KUKA KRL program: MyProgram_242().src

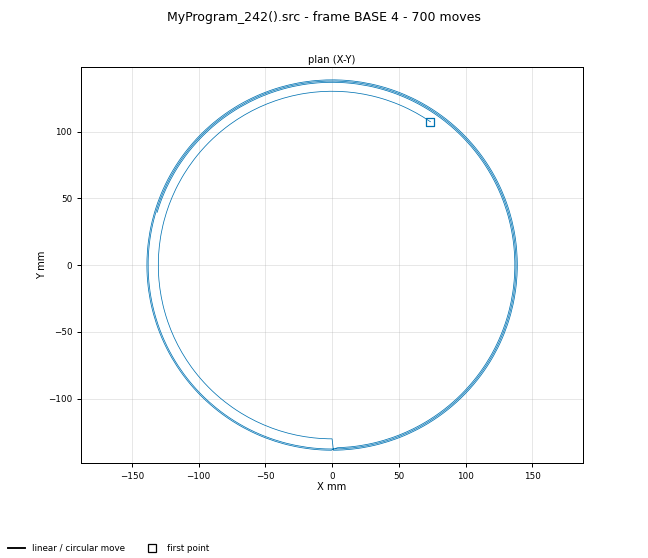
[picture p0: tool path of MyProgram_242().src in frame BASE 4, 700 of 700 moves have a stored position in this frame; points joined in program order, loops and branches not executed]
&ACCESS RVP
&REL 1
&PARAM TEMPLATE = C:\KRC\Roboter\Template\vorgabe
&PARAM EDITMASK = *
DEF MyProgram_242()
; ---- Setting reference (Base) ----
$BASE = BASE_DATA[4]

; --------------------------
; ---- Setting tool (TCP) ----
$TOOL = TOOL_DATA[3]
; --------------------------

$VEL.CP = VEL_APROX_PRINT
Startdeposition()
$VEL.CP = VEL_PRINT
LIN {X 73.6259,Y 107.3159,Z 161,A 55.1179,B 14.0852,C -0.2043,E1 14.1765,E2 754.5488} C_DIS
LIN {X 70.9847,Y 109.081,Z 161,A 56.5627,B 14.0851,C -0.2078,E1 14.1731,E2 753.0982} C_DIS
LIN {X 68.1836,Y 110.8535,Z 161,A 57.9076,B 14.0851,C -0.2066,E1 14.17,E2 751.7664} C_DIS
LIN {X 65.4361,Y 112.4974,Z 161,A 59.3048,B 14.0851,C -0.2083,E1 14.1666,E2 750.3704} C_DIS
LIN {X 62.7519,Y 114.0166,Z 161,A 60.6768,B 14.0851,C -0.2106,E1 14.1633,E2 748.9965} C_DIS
LIN {X 59.8481,Y 115.5669,Z 161,A 62.1112,B 14.0851,C -0.212,E1 14.1597,E2 747.5636} C_DIS
LIN {X 56.9987,Y 116.9979,Z 161,A 63.5064,B 14.085,C -0.2135,E1 14.1562,E2 746.1693} C_DIS
LIN {X 53.5847,Y 118.5997,Z 161,A 65.2897,B 14.085,C -0.2191,E1 14.1517,E2 744.3715} C_DIS
LIN {X 50.1104,Y 120.1079,Z 161,A 66.8675,B 14.085,C -0.2183,E1 14.1476,E2 742.804} C_DIS
LIN {X 46.7383,Y 121.4607,Z 161,A 68.4744,B 14.0849,C -0.2201,E1 14.1434,E2 741.1964} C_DIS
LIN {X 43.7469,Y 122.5698,Z 161,A 69.8364,B 14.0849,C -0.2202,E1 14.1399,E2 739.8394} C_DIS
LIN {X 40.8271,Y 123.5728,Z 161,A 71.1622,B 14.0849,C -0.2204,E1 14.1364,E2 738.5175} C_DIS
LIN {X 37.7836,Y 124.5371,Z 161,A 72.5623,B 14.0849,C -0.2214,E1 14.1327,E2 737.1182} C_DIS
LIN {X 33.9943,Y 125.625,Z 161,A 74.4676,B 14.0848,C -0.2276,E1 14.1275,E2 735.1934} C_DIS
LIN {X 30.0784,Y 126.6195,Z 161,A 76.0649,B 14.0848,C -0.2234,E1 14.1232,E2 733.6176} C_DIS
LIN {X 26.8751,Y 127.3386,Z 161,A 77.4994,B 14.0848,C -0.2239,E1 14.1193,E2 732.1847} C_DIS
LIN {X 23.8559,Y 127.9386,Z 161,A 78.9842,B 14.0848,C -0.2283,E1 14.1152,E2 730.6852} C_DIS
LIN {X 19.9821,Y 128.5993,Z 161,A 80.3539,B 14.0849,C -0.2187,E1 14.1115,E2 729.3576} C_DIS
LIN {X 17.4097,Y 128.9737,Z 161,A 81.7136,B 14.0849,C -0.2252,E1 14.1077,E2 727.9733} C_DIS
LIN {X 14.242,Y 129.3613,Z 161,A 83.119,B 14.0849,C -0.2256,E1 14.1038,E2 726.5684} C_DIS
LIN {X 11.1666,Y 129.6628,Z 161,A 84.5021,B 14.0848,C -0.2265,E1 14.0999,E2 725.1832} C_DIS
LIN {X 7.9833,Y 129.8975,Z 161,A 85.9176,B 14.0848,C -0.2269,E1 14.096,E2 723.767} C_DIS
LIN {X 4.786,Y 130.0549,Z 161,A 87.3094,B 14.0848,C -0.2265,E1 14.0921,E2 722.3779} C_DIS
LIN {X 1.4943,Y 130.1358,Z 161,A 88.733,B 14.0848,C -0.2257,E1 14.0882,E2 720.9579} C_DIS
LIN {X -1.5932,Y 130.1342,Z 161,A 90.1699,B 14.0848,C -0.2278,E1 14.0841,E2 719.5127} C_DIS
LIN {X -5.1925,Y 130.039,Z 161,A 91.6534,B 14.0848,C -0.2246,E1 14.08,E2 718.0418} C_DIS
LIN {X -8.0856,Y 129.8912,Z 161,A 92.9819,B 14.0848,C -0.2258,E1 14.0763,E2 716.7078} C_DIS
LIN {X -11.2683,Y 129.6542,Z 161,A 94.372,B 14.0848,C -0.2249,E1 14.0724,E2 715.3202} C_DIS
LIN {X -14.4438,Y 129.3396,Z 161,A 95.7808,B 14.0848,C -0.2245,E1 14.0685,E2 713.9118} C_DIS
LIN {X -17.6126,Y 128.9471,Z 161,A 97.3138,B 14.0848,C -0.2273,E1 14.0642,E2 712.365} C_DIS
LIN {X -20.6298,Y 128.499,Z 161,A 98.5394,B 14.0848,C -0.2233,E1 14.0609,E2 711.1539} C_DIS
LIN {X -23.9131,Y 127.9277,Z 161,A 100.0038,B 14.0848,C -0.2224,E1 14.0569,E2 709.6908} C_DIS
LIN {X -27.4493,Y 127.2146,Z 161,A 101.5101,B 14.0849,C -0.219,E1 14.0528,E2 708.1949} C_DIS
LIN {X -30.151,Y 126.602,Z 161,A 102.8492,B 14.0849,C -0.2214,E1 14.0491,E2 706.843} C_DIS
LIN {X -33.2702,Y 125.818,Z 161,A 104.3001,B 14.0849,C -0.2212,E1 14.0452,E2 705.3891} C_DIS
LIN {X -36.3399,Y 124.9659,Z 161,A 105.6665,B 14.0849,C -0.2189,E1 14.0415,E2 704.0279} C_DIS
LIN {X -39.3872,Y 124.0391,Z 161,A 107.073,B 14.0849,C -0.2177,E1 14.0378,E2 702.622} C_DIS
LIN {X -42.3168,Y 123.0707,Z 161,A 108.4441,B 14.0849,C -0.2166,E1 14.0341,E2 701.2507} C_DIS
LIN {X -45.3437,Y 121.9879,Z 161,A 109.885,B 14.0849,C -0.2157,E1 14.0304,E2 699.8079} C_DIS
LIN {X -48.4193,Y 120.7999,Z 161,A 111.3149,B 14.0849,C -0.2134,E1 14.0267,E2 698.3819} C_DIS
LIN {X -51.3848,Y 119.5686,Z 161,A 112.7332,B 14.085,C -0.2118,E1 14.023,E2 696.9643} C_DIS
LIN {X -54.2001,Y 118.3196,Z 161,A 114.1986,B 14.085,C -0.213,E1 14.0193,E2 695.4875} C_DIS
LIN {X -57.0785,Y 116.9586,Z 161,A 115.5012,B 14.085,C -0.2084,E1 14.016,E2 694.1977} C_DIS
LIN {X -59.9209,Y 115.5287,Z 161,A 116.919,B 14.085,C -0.2068,E1 14.0125,E2 692.7793} C_DIS
LIN {X -62.7222,Y 114.0331,Z 161,A 118.3262,B 14.0851,C -0.2049,E1 14.009,E2 691.3724} C_DIS
LIN {X -65.5265,Y 112.4451,Z 161,A 119.7877,B 14.0851,C -0.2038,E1 14.0055,E2 689.9074} C_DIS
LIN {X -68.3598,Y 110.7454,Z 161,A 121.3351,B 14.0851,C -0.2039,E1 14.0018,E2 688.3507} C_DIS
LIN {X -71.0666,Y 109.0278,Z 161,A 122.6353,B 14.0852,C -0.1986,E1 13.9988,E2 687.0649} C_DIS
LIN {X -74.0034,Y 107.0567,Z 161,A 124.1527,B 14.0852,C -0.1948,E1 13.9953,E2 685.5537} C_DIS
LIN {X -76.3034,Y 105.4289,Z 161,A 125.5318,B 14.0852,C -0.1962,E1 13.9921,E2 684.1599} C_DIS
LIN {X -79.477,Y 103.0581,Z 161,A 127.3516,B 14.0852,C -0.1949,E1 13.988,E2 682.3333} C_DIS
LIN {X -83.0592,Y 100.193,Z 161,A 129.2786,B 14.0853,C -0.1885,E1 13.9839,E2 680.4192} C_DIS
LIN {X -86.2133,Y 97.4923,Z 161,A 131.2268,B 14.0853,C -0.188,E1 13.9798,E2 678.4592} C_DIS
LIN {X -89.1958,Y 94.7713,Z 161,A 132.9988,B 14.0853,C -0.1841,E1 13.9761,E2 676.6899} C_DIS
LIN {X -92.2874,Y 91.7633,Z 161,A 134.8732,B 14.0855,C -0.1793,E1 13.9724,E2 674.8205} C_DIS
LIN {X -95.3546,Y 88.5719,Z 161,A 136.7631,B 14.0855,C -0.1734,E1 13.9688,E2 672.9397} C_DIS
LIN {X -98.0222,Y 85.6103,Z 161,A 138.665,B 14.0855,C -0.1732,E1 13.9653,E2 671.0229} C_DIS
LIN {X -101.0689,Y 81.9919,Z 161,A 140.6548,B 14.0856,C -0.1659,E1 13.9618,E2 669.0464} C_DIS
LIN {X -103.5133,Y 78.883,Z 161,A 142.367,B 14.0856,C -0.1609,E1 13.9588,E2 667.3397} C_DIS
LIN {X -105.4767,Y 76.2375,Z 161,A 143.8459,B 14.0857,C -0.158,E1 13.9564,E2 665.8592} C_DIS
LIN {X -107.3136,Y 73.6292,Z 161,A 145.2685,B 14.0857,C -0.155,E1 13.9541,E2 664.4363} C_DIS
LIN {X -109.0913,Y 70.9688,Z 161,A 146.6792,B 14.0857,C -0.1514,E1 13.952,E2 663.0271} C_DIS
LIN {X -110.8493,Y 68.1904,Z 161,A 148.1401,B 14.0858,C -0.148,E1 13.9498,E2 661.5664} C_DIS
LIN {X -112.4949,Y 65.4403,Z 161,A 149.6242,B 14.0858,C -0.1462,E1 13.9477,E2 660.0757} C_DIS
LIN {X -114.1557,Y 62.4979,Z 161,A 151.0218,B 14.0858,C -0.1399,E1 13.9458,E2 658.6904} C_DIS
LIN {X -115.5768,Y 59.8291,Z 161,A 152.4245,B 14.0859,C -0.1382,E1 13.944,E2 657.2811} C_DIS
LIN {X -117.0061,Y 56.9822,Z 161,A 153.8389,B 14.0859,C -0.1346,E1 13.9422,E2 655.8671} C_DIS
LIN {X -118.489,Y 53.8322,Z 161,A 155.3666,B 14.0859,C -0.1303,E1 13.9404,E2 654.3419} C_DIS
LIN {X -119.6145,Y 51.2786,Z 161,A 156.6245,B 14.086,C -0.1276,E1 13.939,E2 653.0822} C_DIS
LIN {X -120.8349,Y 48.3325,Z 161,A 158.0533,B 14.086,C -0.1243,E1 13.9375,E2 651.6522} C_DIS
LIN {X -122.019,Y 45.2606,Z 161,A 159.5081,B 14.086,C -0.1203,E1 13.9361,E2 650.1987} C_DIS
LIN {X -123.0645,Y 42.3345,Z 161,A 160.8894,B 14.0861,C -0.1167,E1 13.9348,E2 648.8176} C_DIS
LIN {X -124.0689,Y 39.294,Z 161,A 162.312,B 14.0861,C -0.113,E1 13.9336,E2 647.3953} C_DIS
LIN {X -124.9947,Y 36.2415,Z 161,A 163.8195,B 14.0861,C -0.1115,E1 13.9324,E2 645.8775} C_DIS
LIN {X -125.8456,Y 33.1671,Z 161,A 165.1509,B 14.0861,C -0.1056,E1 13.9315,E2 644.5565} C_DIS
LIN {X -126.6208,Y 30.0728,Z 161,A 166.5675,B 14.0862,C -0.1018,E1 13.9305,E2 643.1402} C_DIS
LIN {X -127.3728,Y 26.717,Z 161,A 168.0921,B 14.0862,C -0.0976,E1 13.9296,E2 641.6164} C_DIS
LIN {X -127.9447,Y 23.8242,Z 161,A 169.4945,B 14.0862,C -0.0964,E1 13.9289,E2 640.2034} C_DIS
LIN {X -128.493,Y 20.668,Z 161,A 170.8524,B 14.0862,C -0.0908,E1 13.9283,E2 638.8534} C_DIS
LIN {X -128.973,Y 17.4148,Z 161,A 172.2813,B 14.0863,C -0.0861,E1 13.9277,E2 637.4285} C_DIS
LIN {X -129.3602,Y 14.2523,Z 161,A 173.7018,B 14.0863,C -0.0823,E1 13.9272,E2 636.0076} C_DIS
LIN {X -129.6614,Y 11.1832,Z 161,A 175.1006,B 14.0863,C -0.0793,E1 13.9269,E2 634.6056} C_DIS
LIN {X -129.8984,Y 7.9682,Z 161,A 176.6346,B 14.0863,C -0.078,E1 13.9266,E2 633.0601} C_DIS
LIN {X -130.1053,Y 3.1501,Z 161,A 178.8132,B 14.0863,C -0.073,E1 13.9264,E2 630.8775} C_DIS
LIN {X -130.1443,Y -0.1417,Z 161,A -179.8418,B 14.0864,C -0.066,E1 13.9264,E2 629.5464} C_DIS
LIN {X -130.0999,Y -3.3439,Z 161,A -178.4539,B 14.0864,C -0.0612,E1 13.9264,E2 628.1627} C_DIS
LIN {X -129.9457,Y -7.1863,Z 161,A -176.5128,B 14.0864,C -0.0625,E1 13.9267,E2 626.1947} C_DIS
LIN {X -129.6591,Y -11.2103,Z 161,A -174.791,B 14.0864,C -0.0558,E1 13.9271,E2 624.4813} C_DIS
LIN {X -129.3395,Y -14.444,Z 161,A -173.4951,B 14.0864,C -0.0481,E1 13.9275,E2 623.2028} C_DIS
LIN {X -128.9453,Y -17.6265,Z 161,A -172.0481,B 14.0865,C -0.0448,E1 13.928,E2 621.7532} C_DIS
LIN {X -128.4921,Y -20.6737,Z 161,A -170.6312,B 14.0865,C -0.0424,E1 13.9286,E2 620.3307} C_DIS
LIN {X -127.9276,Y -23.9136,Z 161,A -169.2425,B 14.0865,C -0.0367,E1 13.9293,E2 618.9505} C_DIS
LIN {X -127.3036,Y -27.0372,Z 161,A -167.7841,B 14.0865,C -0.034,E1 13.9301,E2 617.487} C_DIS
LIN {X -126.5963,Y -30.1746,Z 161,A -166.3629,B 14.0865,C -0.0301,E1 13.931,E2 616.0666} C_DIS
LIN {X -125.8186,Y -33.2682,Z 161,A -164.8112,B 14.0865,C -0.0298,E1 13.9321,E2 614.4991} C_DIS
LIN {X -124.5105,Y -37.8707,Z 161,A -162.6746,B 14.0865,C -0.0246,E1 13.9338,E2 612.3611} C_DIS
LIN {X -123.0627,Y -42.3397,Z 161,A -160.5991,B 14.0865,C -0.019,E1 13.9356,E2 610.2868} C_DIS
LIN {X -121.9873,Y -45.3452,Z 161,A -159.2767,B 14.0865,C -0.013,E1 13.9369,E2 608.9755} C_DIS
LIN {X -120.796,Y -48.4289,Z 161,A -157.8194,B 14.0865,C -0.009,E1 13.9384,E2 607.5193} C_DIS
LIN {X -119.4274,Y -51.7114,Z 161,A -156.3496,B 14.0865,C -0.0023,E1 13.94,E2 606.0621} C_DIS
LIN {X -118.3288,Y -54.1803,Z 161,A -155.0611,B 14.0865,C -0.0017,E1 13.9415,E2 604.7631} C_DIS
LIN {X -116.9719,Y -57.0514,Z 161,A -153.6354,B 14.0865,C 0.0013,E1 13.9432,E2 603.3354} C_DIS
LIN {X -115.5201,Y -59.9372,Z 161,A -152.2025,B 14.0865,C 0.0047,E1 13.945,E2 601.9025} C_DIS
LIN {X -114.0169,Y -62.7514,Z 161,A -150.793,B 14.0865,C 0.0082,E1 13.9469,E2 600.4936} C_DIS
LIN {X -112.4447,Y -65.5272,Z 161,A -149.2073,B 14.0865,C 0.0071,E1 13.9492,E2 598.8876} C_DIS
LIN {X -110.6283,Y -68.5486,Z 161,A -147.8508,B 14.0865,C 0.016,E1 13.9511,E2 597.5554} C_DIS
LIN {X -109.0315,Y -71.0609,Z 161,A -146.4787,B 14.0865,C 0.0176,E1 13.9532,E2 596.1769} C_DIS
LIN {X -107.2589,Y -73.709,Z 161,A -145.0641,B 14.0865,C 0.0207,E1 13.9554,E2 594.762} C_DIS
LIN {X -105.4136,Y -76.3247,Z 161,A -143.6468,B 14.0865,C 0.0238,E1 13.9577,E2 593.3447} C_DIS
LIN {X -103.0905,Y -79.4352,Z 161,A -141.7683,B 14.0865,C 0.0233,E1 13.9609,E2 591.4474} C_DIS
LIN {X -100.5997,Y -82.5666,Z 161,A -140.0952,B 14.0865,C 0.0296,E1 13.9638,E2 589.7859} C_DIS
LIN {X -97.9974,Y -85.6387,Z 161,A -138.3713,B 14.0865,C 0.0347,E1 13.9669,E2 588.0687} C_DIS
LIN {X -95.8775,Y -88.0056,Z 161,A -136.798,B 14.0865,C 0.0331,E1 13.9699,E2 586.4756} C_DIS
LIN {X -92.6228,Y -91.4257,Z 161,A -134.8322,B 14.0865,C 0.0404,E1 13.9737,E2 584.5242} C_DIS
LIN {X -89.7209,Y -94.2747,Z 161,A -132.8894,B 14.0865,C 0.0398,E1 13.9777,E2 582.5643} C_DIS
LIN {X -86.8005,Y -96.9698,Z 161,A -131.2805,B 14.0865,C 0.047,E1 13.981,E2 580.9727} C_DIS
LIN {X -83.8113,Y -99.5649,Z 161,A -129.3858,B 14.0865,C 0.0461,E1 13.985,E2 579.0608} C_DIS
LIN {X -80.1295,Y -102.5517,Z 161,A -127.4162,B 14.0865,C 0.0529,E1 13.9893,E2 577.1058} C_DIS
LIN {X -77.5216,Y -104.5367,Z 161,A -125.9765,B 14.0865,C 0.0554,E1 13.9925,E2 575.667} C_DIS
LIN {X -74.9412,Y -106.4016,Z 161,A -124.5698,B 14.0865,C 0.0576,E1 13.9957,E2 574.2602} C_DIS
LIN {X -71.6886,Y -108.6197,Z 161,A -122.6855,B 14.0865,C 0.0562,E1 14.0001,E2 572.3583} C_DIS
LIN {X -68.1778,Y -110.8571,Z 161,A -120.9872,B 14.0865,C 0.0625,E1 14.0041,E2 570.6765} C_DIS
LIN {X -65.4414,Y -112.4943,Z 161,A -119.5778,B 14.0865,C 0.0643,E1 14.0075,E2 569.2667} C_DIS
LIN {X -62.7563,Y -114.0142,Z 161,A -118.1916,B 14.0865,C 0.0654,E1 14.0109,E2 567.8774} C_DIS
LIN {X -59.8522,Y -115.5647,Z 161,A -116.7433,B 14.0865,C 0.0672,E1 14.0144,E2 566.4294} C_DIS
LIN {X -57.0023,Y -116.9962,Z 161,A -115.3347,B 14.0865,C 0.0688,E1 14.018,E2 565.0203} C_DIS
LIN {X -53.636,Y -118.5767,Z 161,A -113.7967,B 14.0864,C 0.0734,E1 14.0218,E2 563.4942} C_DIS
LIN {X -51.2692,Y -119.6186,Z 161,A -112.5522,B 14.0864,C 0.0716,E1 14.0251,E2 562.2372} C_DIS
LIN {X -47.7588,Y -121.064,Z 161,A -110.9356,B 14.0864,C 0.0748,E1 14.0292,E2 560.6271} C_DIS
LIN {X -44.8477,Y -122.173,Z 161,A -109.519,B 14.0864,C 0.0748,E1 14.0329,E2 559.2051} C_DIS
LIN {X -42.3399,Y -123.0627,Z 161,A -108.3263,B 14.0864,C 0.0752,E1 14.0361,E2 558.0097} C_DIS
LIN {X -39.3122,Y -124.063,Z 161,A -106.9169,B 14.0864,C 0.0762,E1 14.0398,E2 556.5995} C_DIS
LIN {X -36.2456,Y -124.9935,Z 161,A -105.4997,B 14.0864,C 0.077,E1 14.0436,E2 555.1814} C_DIS
LIN {X -33.1768,Y -125.843,Z 161,A -104.1015,B 14.0864,C 0.078,E1 14.0474,E2 553.7834} C_DIS
LIN {X -30.0897,Y -126.6168,Z 161,A -102.6988,B 14.0864,C 0.0787,E1 14.0512,E2 552.3803} C_DIS
LIN {X -26.8938,Y -127.3346,Z 161,A -101.262,B 14.0864,C 0.0796,E1 14.0551,E2 550.9438} C_DIS
LIN {X -23.2646,Y -128.0466,Z 161,A -99.7802,B 14.0864,C 0.0844,E1 14.0592,E2 549.4791} C_DIS
LIN {X -20.6714,Y -128.4925,Z 161,A -98.4478,B 14.0864,C 0.0799,E1 14.0629,E2 548.1257} C_DIS
LIN {X -17.411,Y -128.9735,Z 161,A -97.0294,B 14.0864,C 0.0812,E1 14.0668,E2 546.7106} C_DIS
LIN {X -14.2422,Y -129.3612,Z 161,A -95.4636,B 14.0864,C 0.0769,E1 14.0712,E2 545.1252} C_DIS
LIN {X -9.5785,Y -129.7896,Z 161,A -93.5043,B 14.0864,C 0.08,E1 14.0766,E2 543.1773} C_DIS
LIN {X -6.2811,Y -129.9912,Z 161,A -92.1053,B 14.0864,C 0.0817,E1 14.0805,E2 541.7844} C_DIS
LIN {X -3.0902,Y -130.107,Z 161,A -90.699,B 14.0864,C 0.0816,E1 14.0844,E2 540.3774} C_DIS
LIN {X -0.0064,Y -130.1446,Z 161,A -89.2963,B 14.0864,C 0.0801,E1 14.0884,E2 538.9687} C_DIS
LIN {X -0.0064,Y -130.1446,Z 161,A -89.2963,B 14.0864,C 0.0801,E1 14.0884,E2 538.9687} C_DIS
Enddeposition()
LIN {X 0.9753,Y -138.6804,Z 162,A -92.6437,B 24.9722,C -1.2174,E1 25.001,E2 539.3993} C_DIS
Startdeposition()
$VEL.CP = VEL_PRINT
LIN {X 3.7085,Y -138.6375,Z 162,A -90.9723,B 24.9708,C -1.2478,E1 25.0059,E2 537.6562} C_DIS
LIN {X 8.2859,Y -138.4394,Z 162,A -88.9916,B 24.9706,C -1.2535,E1 25.0114,E2 535.6628} C_DIS
LIN {X 14.8199,Y -137.8928,Z 162,A -86.3827,B 24.9708,C -1.2494,E1 25.0186,E2 533.0653} C_DIS
LIN {X 19.2083,Y -137.3508,Z 162,A -84.5954,B 24.9708,C -1.2483,E1 25.0236,E2 531.2819} C_DIS
LIN {X 22.4873,Y -136.852,Z 162,A -83.2381,B 24.9708,C -1.2486,E1 25.0273,E2 529.9251} C_DIS
LIN {X 28.0328,Y -135.8246,Z 162,A -80.8102,B 24.9704,C -1.2562,E1 25.034,E2 527.4823} C_DIS
LIN {X 32.1897,Y -134.8997,Z 162,A -79.1481,B 24.9706,C -1.2524,E1 25.0385,E2 525.8314} C_DIS
LIN {X 35.5715,Y -134.0473,Z 162,A -77.6983,B 24.9706,C -1.2544,E1 25.0424,E2 524.3791} C_DIS
LIN {X 39.11,Y -133.0579,Z 162,A -76.2619,B 24.9706,C -1.2515,E1 25.0463,E2 522.9519} C_DIS
LIN {X 42.0399,Y -132.1614,Z 162,A -75.0069,B 24.9706,C -1.2525,E1 25.0496,E2 521.697} C_DIS
LIN {X 45.6855,Y -130.9461,Z 162,A -73.6635,B 24.9712,C -1.2407,E1 25.0531,E2 520.3841} C_DIS
LIN {X 48.0279,Y -130.1065,Z 162,A -72.2874,B 24.9702,C -1.2618,E1 25.0568,E2 518.9609} C_DIS
LIN {X 51.3498,Y -128.831,Z 162,A -70.9235,B 24.9704,C -1.2579,E1 25.0603,E2 517.6094} C_DIS
LIN {X 54.6499,Y -127.4657,Z 162,A -69.429,B 24.9702,C -1.2612,E1 25.0642,E2 516.1105} C_DIS
LIN {X 57.9984,Y -125.9769,Z 162,A -67.9996,B 24.9703,C -1.2587,E1 25.0678,E2 514.6904} C_DIS
LIN {X 61.0435,Y -124.53,Z 162,A -66.5311,B 24.97,C -1.2654,E1 25.0715,E2 513.2101} C_DIS
LIN {X 63.9672,Y -123.0547,Z 162,A -65.1072,B 24.9697,C -1.2718,E1 25.0751,E2 511.775} C_DIS
LIN {X 67.9591,Y -120.8968,Z 162,A -63.229,B 24.9695,C -1.2754,E1 25.0797,E2 509.8938} C_DIS
LIN {X 71.8296,Y -118.6381,Z 162,A -61.3598,B 24.9693,C -1.2799,E1 25.0842,E2 508.0197} C_DIS
LIN {X 75.7781,Y -116.1561,Z 162,A -59.4156,B 24.9691,C -1.2847,E1 25.0888,E2 506.0703} C_DIS
LIN {X 79.6326,Y -113.5485,Z 162,A -57.504,B 24.9689,C -1.2881,E1 25.0932,E2 504.1573} C_DIS
LIN {X 83.0656,Y -111.0616,Z 162,A -55.7626,B 24.9688,C -1.2913,E1 25.0971,E2 502.4146} C_DIS
LIN {X 86.6721,Y -108.2708,Z 162,A -53.9067,B 24.9686,C -1.2939,E1 25.1011,E2 500.5595} C_DIS
LIN {X 90.2073,Y -105.3436,Z 162,A -52.1152,B 24.9687,C -1.2922,E1 25.105,E2 498.7788} C_DIS
LIN {X 93.3673,Y -102.5528,Z 162,A -50.2808,B 24.9683,C -1.3018,E1 25.1088,E2 496.9292} C_DIS
LIN {X 96.8454,Y -99.2752,Z 162,A -48.3436,B 24.9681,C -1.3045,E1 25.1127,E2 494.9937} C_DIS
LIN {X 99.9045,Y -96.1962,Z 162,A -46.6208,B 24.9681,C -1.305,E1 25.1161,E2 493.2772} C_DIS
LIN {X 102.8585,Y -93.0304,Z 162,A -44.7439,B 24.9676,C -1.3148,E1 25.1196,E2 491.3854} C_DIS
LIN {X 105.9921,Y -89.4444,Z 162,A -42.8137,B 24.9675,C -1.3178,E1 25.1231,E2 489.4567} C_DIS
LIN {X 108.8664,Y -85.9226,Z 162,A -40.9278,B 24.9672,C -1.3235,E1 25.1264,E2 487.5664} C_DIS
LIN {X 111.3769,Y -82.6421,Z 162,A -39.2245,B 24.967,C -1.328,E1 25.1293,E2 485.8604} C_DIS
LIN {X 113.7244,Y -79.3806,Z 162,A -37.6296,B 24.967,C -1.329,E1 25.1319,E2 484.2711} C_DIS
LIN {X 116.1586,Y -75.7744,Z 162,A -35.8119,B 24.9666,C -1.3353,E1 25.1347,E2 482.4473} C_DIS
LIN {X 118.5147,Y -72.0336,Z 162,A -34.0007,B 24.9664,C -1.3398,E1 25.1373,E2 480.6348} C_DIS
LIN {X 120.7254,Y -68.2641,Z 162,A -32.2065,B 24.9661,C -1.3446,E1 25.1398,E2 478.8387} C_DIS
LIN {X 122.8089,Y -64.4352,Z 162,A -30.5511,B 24.9663,C -1.3416,E1 25.142,E2 477.199} C_DIS
LIN {X 124.191,Y -61.7308,Z 162,A -29.3366,B 24.9663,C -1.3431,E1 25.1435,E2 475.9875} C_DIS
LIN {X 125.746,Y -58.4976,Z 162,A -27.988,B 24.9663,C -1.3399,E1 25.1451,E2 474.6537} C_DIS
LIN {X 127.389,Y -54.8273,Z 162,A -26.1614,B 24.9656,C -1.3547,E1 25.1472,E2 472.802} C_DIS
LIN {X 128.7705,Y -51.5,Z 162,A -24.6262,B 24.9652,C -1.3622,E1 25.1488,E2 471.2577} C_DIS
LIN {X 130.3355,Y -47.4,Z 162,A -22.8953,B 24.9652,C -1.3632,E1 25.1505,E2 469.5342} C_DIS
LIN {X 131.3138,Y -44.6245,Z 162,A -21.5185,B 24.9645,C -1.3765,E1 25.1518,E2 468.1337} C_DIS
LIN {X 132.6699,Y -40.4067,Z 162,A -19.8106,B 24.9645,C -1.3753,E1 25.1532,E2 466.4384} C_DIS
LIN {X 133.7855,Y -36.5526,Z 162,A -18.0491,B 24.964,C -1.3868,E1 25.1545,E2 464.66} C_DIS
LIN {X 135.5398,Y -29.3766,Z 162,A -15.2875,B 24.9643,C -1.3797,E1 25.1563,E2 461.931} C_DIS
LIN {X 136.5038,Y -24.5099,Z 162,A -13.0623,B 24.9635,C -1.3968,E1 25.1575,E2 459.6785} C_DIS
LIN {X 137.461,Y -18.4024,Z 162,A -10.5107,B 24.963,C -1.4051,E1 25.1586,E2 457.1223} C_DIS
LIN {X 137.9164,Y -14.6005,Z 162,A -9.0149,B 24.963,C -1.4053,E1 25.159,E2 455.6348} C_DIS
LIN {X 138.2749,Y -10.6987,Z 162,A -7.3449,B 24.9626,C -1.4137,E1 25.1594,E2 453.9549} C_DIS
LIN {X 138.4663,Y -7.8494,Z 162,A -6.0652,B 24.962,C -1.4235,E1 25.1596,E2 452.6597} C_DIS
LIN {X 138.6555,Y -3.0458,Z 162,A -4.1721,B 24.962,C -1.4247,E1 25.1598,E2 450.7752} C_DIS
LIN {X 138.6846,Y 0.9336,Z 162,A -2.5259,B 24.9617,C -1.4303,E1 25.1598,E2 449.1256} C_DIS
LIN {X 138.5957,Y 5.0433,Z 162,A -0.7011,B 24.961,C -1.4434,E1 25.1596,E2 447.2808} C_DIS
LIN {X 138.1484,Y 12.2225,Z 162,A 2.1078,B 24.961,C -1.4436,E1 25.159,E2 444.4881} C_DIS
LIN {X 137.7591,Y 16.0201,Z 162,A 3.6244,B 24.9609,C -1.4452,E1 25.1586,E2 442.9766} C_DIS
LIN {X 137.2957,Y 19.5936,Z 162,A 5.4378,B 24.9596,C -1.4692,E1 25.1579,E2 441.1174} C_DIS
LIN {X 136.6815,Y 23.5089,Z 162,A 6.7441,B 24.9603,C -1.455,E1 25.1573,E2 439.8522} C_DIS
LIN {X 136.0133,Y 27.1056,Z 162,A 8.2737,B 24.96,C -1.461,E1 25.1565,E2 438.3175} C_DIS
LIN {X 135.2956,Y 30.4839,Z 162,A 9.586,B 24.9601,C -1.4588,E1 25.1557,E2 437.0179} C_DIS
LIN {X 134.5402,Y 33.6623,Z 162,A 10.9233,B 24.9599,C -1.4624,E1 25.1548,E2 435.6799} C_DIS
LIN {X 133.7126,Y 36.8137,Z 162,A 12.2469,B 24.9598,C -1.4654,E1 25.1538,E2 434.3569} C_DIS
LIN {X 132.8113,Y 39.9448,Z 162,A 13.6471,B 24.9594,C -1.4727,E1 25.1527,E2 432.9474} C_DIS
LIN {X 131.8109,Y 43.1321,Z 162,A 14.9339,B 24.9594,C -1.4716,E1 25.1516,E2 431.6707} C_DIS
LIN {X 130.6246,Y 46.598,Z 162,A 16.4084,B 24.9594,C -1.474,E1 25.1503,E2 430.1988} C_DIS
LIN {X 129.3548,Y 50.0134,Z 162,A 18.0698,B 24.9585,C -1.4876,E1 25.1486,E2 428.5144} C_DIS
LIN {X 127.9962,Y 53.3939,Z 162,A 19.4247,B 24.9588,C -1.4834,E1 25.1472,E2 427.177} C_DIS
LIN {X 126.8443,Y 56.0786,Z 162,A 20.6478,B 24.9585,C -1.4879,E1 25.1458,E2 425.9499} C_DIS
LIN {X 125.4423,Y 59.1495,Z 162,A 22.1319,B 24.958,C -1.4972,E1 25.1441,E2 424.452} C_DIS
LIN {X 123.9038,Y 62.3077,Z 162,A 23.4532,B 24.9582,C -1.4938,E1 25.1424,E2 423.1457} C_DIS
LIN {X 122.0968,Y 65.779,Z 162,A 25.225,B 24.9574,C -1.5074,E1 25.1401,E2 421.3512} C_DIS
LIN {X 119.8214,Y 69.8389,Z 162,A 27.1533,B 24.9571,C -1.5131,E1 25.1374,E2 419.4195} C_DIS
LIN {X 117.384,Y 73.8614,Z 162,A 28.9985,B 24.9571,C -1.5127,E1 25.1347,E2 417.5846} C_DIS
LIN {X 115.1906,Y 77.2377,Z 162,A 30.6508,B 24.9569,C -1.5165,E1 25.1322,E2 415.9316} C_DIS
LIN {X 112.8106,Y 80.6736,Z 162,A 32.3991,B 24.9566,C -1.5222,E1 25.1294,E2 414.1783} C_DIS
LIN {X 110.2402,Y 84.1521,Z 162,A 34.1841,B 24.9563,C -1.5266,E1 25.1264,E2 412.3914} C_DIS
LIN {X 107.5398,Y 87.5769,Z 162,A 35.9758,B 24.9561,C -1.5305,E1 25.1232,E2 410.5989} C_DIS
LIN {X 104.687,Y 90.968,Z 162,A 37.8485,B 24.9557,C -1.5373,E1 25.1198,E2 408.7186} C_DIS
LIN {X 101.5212,Y 94.4877,Z 162,A 39.7526,B 24.9557,C -1.5389,E1 25.1162,E2 406.8193} C_DIS
LIN {X 98.4714,Y 97.662,Z 162,A 41.5766,B 24.9554,C -1.5432,E1 25.1127,E2 404.9928} C_DIS
LIN {X 95.1807,Y 100.8717,Z 162,A 43.4532,B 24.9552,C -1.546,E1 25.1089,E2 403.1173} C_DIS
LIN {X 91.9435,Y 103.831,Z 162,A 45.1593,B 24.9553,C -1.5438,E1 25.1054,E2 401.4234} C_DIS
LIN {X 88.9102,Y 106.4403,Z 162,A 46.9207,B 24.9548,C -1.5532,E1 25.1016,E2 399.6466} C_DIS
LIN {X 85.4258,Y 109.2566,Z 162,A 48.7513,B 24.9547,C -1.5556,E1 25.0976,E2 397.8172} C_DIS
LIN {X 81.956,Y 111.8826,Z 162,A 50.5337,B 24.9545,C -1.558,E1 25.0936,E2 396.0354} C_DIS
LIN {X 78.3975,Y 114.4042,Z 162,A 52.2951,B 24.9545,C -1.5589,E1 25.0896,E2 394.2781} C_DIS
LIN {X 74.835,Y 116.7656,Z 162,A 54.0846,B 24.9542,C -1.5631,E1 25.0854,E2 392.4844} C_DIS
LIN {X 71.4071,Y 118.8936,Z 162,A 55.799,B 24.9539,C -1.5684,E1 25.0813,E2 390.763} C_DIS
LIN {X 67.3342,Y 121.2461,Z 162,A 57.7096,B 24.9539,C -1.5694,E1 25.0766,E2 388.8556} C_DIS
LIN {X 63.1987,Y 123.4502,Z 162,A 59.5084,B 24.9541,C -1.5644,E1 25.0722,E2 387.0738} C_DIS
LIN {X 60.1258,Y 124.9758,Z 162,A 61.0447,B 24.9536,C -1.5728,E1 25.0683,E2 385.5215} C_DIS
LIN {X 54.0838,Y 127.7081,Z 162,A 63.7749,B 24.9535,C -1.5755,E1 25.0614,E2 382.7917} C_DIS
LIN {X 50.8184,Y 129.0419,Z 162,A 65.0541,B 24.954,C -1.5671,E1 25.0581,E2 381.5354} C_DIS
LIN {X 47.3828,Y 130.3417,Z 162,A 66.5859,B 24.9539,C -1.5694,E1 25.0541,E2 380.0014} C_DIS
LIN {X 44.0908,Y 131.4916,Z 162,A 68.0823,B 24.9536,C -1.5737,E1 25.0501,E2 378.4976} C_DIS
LIN {X 40.3711,Y 132.6808,Z 162,A 69.7223,B 24.9534,C -1.5765,E1 25.0457,E2 376.8539} C_DIS
LIN {X 36.2698,Y 133.8611,Z 162,A 71.4565,B 24.9534,C -1.5761,E1 25.0411,E2 375.1235} C_DIS
LIN {X 33.1096,Y 134.6779,Z 162,A 72.7978,B 24.9534,C -1.5766,E1 25.0375,E2 373.7832} C_DIS
LIN {X 29.5481,Y 135.5027,Z 162,A 74.3494,B 24.9532,C -1.5797,E1 25.0332,E2 372.2263} C_DIS
LIN {X 22.0964,Y 136.9172,Z 162,A 77.6119,B 24.9528,C -1.588,E1 25.0242,E2 368.9478} C_DIS
LIN {X 18.3128,Y 137.4728,Z 162,A 79.0783,B 24.9531,C -1.5822,E1 25.0202,E2 367.4964} C_DIS
LIN {X 15.3307,Y 137.8378,Z 162,A 80.4516,B 24.9527,C -1.5896,E1 25.0163,E2 366.1064} C_DIS
LIN {X 10.2761,Y 138.3058,Z 162,A 82.2843,B 24.9535,C -1.5753,E1 25.0113,E2 364.3087} C_DIS
LIN {X 6.9774,Y 138.5113,Z 162,A 83.8133,B 24.953,C -1.5843,E1 25.007,E2 362.759} C_DIS
LIN {X 1.7495,Y 138.6771,Z 162,A 86.066,B 24.9527,C -1.589,E1 25.0007,E2 360.4956} C_DIS
LIN {X -4.377,Y 138.6189,Z 162,A 88.4104,B 24.9533,C -1.5782,E1 24.9942,E2 358.1767} C_DIS
LIN {X -8.2135,Y 138.4439,Z 162,A 90.073,B 24.9531,C -1.5817,E1 24.9896,E2 356.5051} C_DIS
LIN {X -11.2796,Y 138.228,Z 162,A 91.3447,B 24.9531,C -1.5812,E1 24.986,E2 355.2341} C_DIS
LIN {X -15.2031,Y 137.8515,Z 162,A 92.9131,B 24.9534,C -1.5771,E1 24.9817,E2 353.6745} C_DIS
LIN {X -21.8317,Y 136.9591,Z 162,A 95.8247,B 24.953,C -1.5832,E1 24.9736,E2 350.746} C_DIS
LIN {X -25.8999,Y 136.2469,Z 162,A 97.3948,B 24.9535,C -1.5746,E1 24.9693,E2 349.1949} C_DIS
LIN {X -29.2592,Y 135.5651,Z 162,A 98.7912,B 24.9537,C -1.5723,E1 24.9655,E2 347.8022} C_DIS
LIN {X -32.4537,Y 134.836,Z 162,A 100.1428,B 24.9537,C -1.5709,E1 24.9619,E2 346.4521} C_DIS
LIN {X -35.5954,Y 134.0409,Z 162,A 101.4816,B 24.9538,C -1.5695,E1 24.9582,E2 345.1146} C_DIS
LIN {X -38.5099,Y 133.2336,Z 162,A 102.8193,B 24.9536,C -1.5729,E1 24.9546,E2 343.7668} C_DIS
LIN {X -42.4162,Y 132.0412,Z 162,A 104.4798,B 24.9538,C -1.5694,E1 24.9502,E2 342.1116} C_DIS
LIN {X -46.2608,Y 130.7462,Z 162,A 106.2062,B 24.9538,C -1.57,E1 24.9456,E2 340.3806} C_DIS
LIN {X -52.9314,Y 128.1894,Z 162,A 109.1368,B 24.9541,C -1.5647,E1 24.938,E2 337.4561} C_DIS
LIN {X -55.93,Y 126.9108,Z 162,A 110.4245,B 24.9544,C -1.5596,E1 24.9348,E2 336.1776} C_DIS
LIN {X -59.4666,Y 125.2908,Z 162,A 112.0823,B 24.9544,C -1.5597,E1 24.9306,E2 334.5153} C_DIS
LIN {X -63.2797,Y 123.4089,Z 162,A 114.0981,B 24.9538,C -1.5705,E1 24.9255,E2 332.4684} C_DIS
LIN {X -66.2568,Y 121.8382,Z 162,A 115.2476,B 24.9547,C -1.5553,E1 24.9227,E2 331.3519} C_DIS
LIN {X -69.8279,Y 119.8278,Z 162,A 117.0058,B 24.9547,C -1.5556,E1 24.9184,E2 329.5877} C_DIS
LIN {X -72.8832,Y 117.9945,Z 162,A 118.5463,B 24.9547,C -1.5564,E1 24.9148,E2 328.0405} C_DIS
LIN {X -76.9712,Y 115.3686,Z 162,A 120.5028,B 24.955,C -1.5498,E1 24.9102,E2 326.0934} C_DIS
LIN {X -80.7672,Y 112.7437,Z 162,A 122.4166,B 24.9552,C -1.5462,E1 24.9058,E2 324.1816} C_DIS
LIN {X -84.3925,Y 110.0564,Z 162,A 124.2857,B 24.9554,C -1.5424,E1 24.9017,E2 322.3147} C_DIS
LIN {X -88.0186,Y 107.1788,Z 162,A 126.1283,B 24.9559,C -1.5345,E1 24.8977,E2 320.4841} C_DIS
LIN {X -91.163,Y 104.5169,Z 162,A 127.9255,B 24.9559,C -1.5355,E1 24.8939,E2 318.6775} C_DIS
LIN {X -94.6537,Y 101.3666,Z 162,A 129.8974,B 24.956,C -1.5324,E1 24.8898,E2 316.7049} C_DIS
LIN {X -98.0615,Y 98.0745,Z 162,A 131.8916,B 24.9562,C -1.5295,E1 24.8858,E2 314.7094} C_DIS
LIN {X -101.3864,Y 94.6324,Z 162,A 133.84,B 24.9565,C -1.523,E1 24.8821,E2 312.768} C_DIS
LIN {X -104.514,Y 91.1663,Z 162,A 135.7797,B 24.9568,C -1.5185,E1 24.8785,E2 310.8303} C_DIS
LIN {X -107.4685,Y 87.6642,Z 162,A 137.6801,B 24.9571,C -1.5138,E1 24.8751,E2 308.9323} C_DIS
LIN {X -110.2583,Y 84.1285,Z 162,A 139.526,B 24.9574,C -1.5079,E1 24.872,E2 307.0916} C_DIS
LIN {X -112.8305,Y 80.6459,Z 162,A 141.1723,B 24.9581,C -1.4955,E1 24.8693,E2 305.4667} C_DIS
LIN {X -114.757,Y 77.8802,Z 162,A 143.0753,B 24.9568,C -1.518,E1 24.8662,E2 303.5009} C_DIS
LIN {X -116.9809,Y 74.4987,Z 162,A 144.8244,B 24.9568,C -1.5171,E1 24.8636,E2 301.7449} C_DIS
LIN {X -119.2774,Y 70.7633,Z 162,A 146.1698,B 24.9585,C -1.4876,E1 24.8618,E2 300.4628} C_DIS
LIN {X -121.0636,Y 67.6623,Z 162,A 147.7337,B 24.9585,C -1.4876,E1 24.8596,E2 298.8908} C_DIS
LIN {X -123.1055,Y 63.8703,Z 162,A 149.5097,B 24.9588,C -1.4821,E1 24.8573,E2 297.1186} C_DIS
LIN {X -124.8322,Y 60.4264,Z 162,A 150.9827,B 24.9595,C -1.4711,E1 24.8555,E2 295.6638} C_DIS
LIN {X -126.4561,Y 56.9466,Z 162,A 152.6326,B 24.9595,C -1.4695,E1 24.8536,E2 294.0088} C_DIS
LIN {X -128.0741,Y 53.2074,Z 162,A 155.2849,B 24.957,C -1.5144,E1 24.8506,E2 291.2346} C_DIS
LIN {X -130.5722,Y 46.7435,Z 162,A 157.2578,B 24.9601,C -1.4591,E1 24.8488,E2 289.3824} C_DIS
LIN {X -132.0016,Y 42.5404,Z 162,A 159.0595,B 24.9605,C -1.4515,E1 24.8472,E2 287.5885} C_DIS
LIN {X -133.1463,Y 38.808,Z 162,A 160.6758,B 24.9608,C -1.4465,E1 24.8459,E2 285.9749} C_DIS
LIN {X -134.0231,Y 35.6622,Z 162,A 162.0097,B 24.9611,C -1.4413,E1 24.845,E2 284.6456} C_DIS
LIN {X -134.7841,Y 32.6691,Z 162,A 163.4131,B 24.961,C -1.4436,E1 24.844,E2 283.2284} C_DIS
LIN {X -135.8024,Y 28.1419,Z 162,A 165.2493,B 24.9615,C -1.4332,E1 24.8429,E2 281.4063} C_DIS
LIN {X -136.5108,Y 24.4708,Z 162,A 166.7998,B 24.9618,C -1.4284,E1 24.8421,E2 279.858} C_DIS
LIN {X -137.0751,Y 21.0822,Z 162,A 168.2225,B 24.962,C -1.4239,E1 24.8415,E2 278.4376} C_DIS
LIN {X -137.5325,Y 17.8573,Z 162,A 169.5741,B 24.9622,C -1.4197,E1 24.841,E2 277.0879} C_DIS
LIN {X -137.9119,Y 14.6426,Z 162,A 170.9259,B 24.9624,C -1.416,E1 24.8406,E2 275.7368} C_DIS
LIN {X -138.2715,Y 10.7463,Z 162,A 172.6664,B 24.9624,C -1.417,E1 24.8402,E2 273.9835} C_DIS
LIN {X -138.6134,Y 4.5475,Z 162,A 175.0613,B 24.9633,C -1.3997,E1 24.8399,E2 271.6154} C_DIS
LIN {X -138.6844,Y -0.9781,Z 162,A 177.4806,B 24.9633,C -1.3991,E1 24.8399,E2 269.183} C_DIS
LIN {X -138.6093,Y -4.6957,Z 162,A 178.9811,B 24.9637,C -1.3921,E1 24.8399,E2 267.6899} C_DIS
LIN {X -138.4586,Y -7.9736,Z 162,A -179.6455,B 24.9639,C -1.3886,E1 24.8401,E2 266.3168} C_DIS
LIN {X -138.1793,Y -11.8566,Z 162,A -177.951,B 24.9639,C -1.3877,E1 24.8405,E2 264.6141} C_DIS
LIN {X -137.7394,Y -16.1848,Z 162,A -176.2257,B 24.9644,C -1.3781,E1 24.841,E2 262.9014} C_DIS
LIN {X -137.311,Y -19.4866,Z 162,A -174.8193,B 24.9646,C -1.3752,E1 24.8415,E2 261.4935} C_DIS
LIN {X -136.7858,Y -22.8838,Z 162,A -173.413,B 24.9648,C -1.3699,E1 24.8422,E2 260.0914} C_DIS
LIN {X -136.2043,Y -26.1227,Z 162,A -172.0713,B 24.9651,C -1.3646,E1 24.8428,E2 258.7545} C_DIS
LIN {X -135.5995,Y -29.1,Z 162,A -170.8014,B 24.9653,C -1.3614,E1 24.8436,E2 257.4848} C_DIS
LIN {X -134.7448,Y -32.8322,Z 162,A -169.093,B 24.9653,C -1.3628,E1 24.8447,E2 255.7629} C_DIS
LIN {X -133.7365,Y -36.7282,Z 162,A -167.4885,B 24.9656,C -1.3546,E1 24.8458,E2 254.1687} C_DIS
LIN {X -131.6189,Y -43.7085,Z 162,A -164.4954,B 24.9662,C -1.3441,E1 24.8483,E2 251.1833} C_DIS
LIN {X -130.309,Y -47.4736,Z 162,A -162.6604,B 24.9659,C -1.3488,E1 24.85,E2 249.3267} C_DIS
LIN {X -128.839,Y -51.33,Z 162,A -161.1072,B 24.9666,C -1.3358,E1 24.8516,E2 247.7958} C_DIS
LIN {X -127.5804,Y -54.3845,Z 162,A -159.6118,B 24.9664,C -1.3385,E1 24.8532,E2 246.2857} C_DIS
LIN {X -125.6973,Y -58.603,Z 162,A -157.7589,B 24.9669,C -1.33,E1 24.8554,E2 244.4428} C_DIS
LIN {X -123.8557,Y -62.4021,Z 162,A -156.1411,B 24.9674,C -1.3184,E1 24.8573,E2 242.8439} C_DIS
LIN {X -121.953,Y -66.0464,Z 162,A -154.2538,B 24.9672,C -1.3234,E1 24.8598,E2 240.9348} C_DIS
LIN {X -119.9426,Y -69.6295,Z 162,A -152.6051,B 24.9676,C -1.3162,E1 24.8621,E2 239.2946} C_DIS
LIN {X -117.7872,Y -73.2165,Z 162,A -150.8117,B 24.9676,C -1.3149,E1 24.8647,E2 237.4952} C_DIS
LIN {X -116.1998,Y -75.7108,Z 162,A -149.4463,B 24.9674,C -1.3191,E1 24.8668,E2 236.1127} C_DIS
LIN {X -113.3389,Y -79.9298,Z 162,A -147.4294,B 24.9679,C -1.309,E1 24.87,E2 234.11} C_DIS
LIN {X -111.373,Y -82.6473,Z 162,A -146.0297,B 24.968,C -1.3062,E1 24.8723,E2 232.7102} C_DIS
LIN {X -108.5026,Y -86.3809,Z 162,A -144.1671,B 24.9685,C -1.297,E1 24.8755,E2 230.8607} C_DIS
LIN {X -105.8207,Y -89.6466,Z 162,A -142.4133,B 24.9687,C -1.2932,E1 24.8786,E2 229.1079} C_DIS
LIN {X -103.2945,Y -92.5457,Z 162,A -140.7564,B 24.9687,C -1.2931,E1 24.8817,E2 227.4438} C_DIS
LIN {X -100.2435,Y -95.8421,Z 162,A -138.9951,B 24.9691,C -1.2839,E1 24.8851,E2 225.6966} C_DIS
LIN {X -97.5557,Y -98.577,Z 162,A -137.3206,B 24.9691,C -1.2852,E1 24.8884,E2 224.012} C_DIS
LIN {X -94.5331,Y -101.4789,Z 162,A -135.5605,B 24.9691,C -1.2831,E1 24.8919,E2 222.2497} C_DIS
LIN {X -91.0071,Y -104.6529,Z 162,A -133.6106,B 24.9694,C -1.2785,E1 24.896,E2 220.3029} C_DIS
LIN {X -87.8601,Y -107.3084,Z 162,A -131.9192,B 24.9696,C -1.2747,E1 24.8996,E2 218.6141} C_DIS
LIN {X -84.799,Y -109.7435,Z 162,A -130.3085,B 24.9697,C -1.2714,E1 24.9032,E2 217.0053} C_DIS
LIN {X -81.2961,Y -112.3629,Z 162,A -128.4852,B 24.9698,C -1.269,E1 24.9073,E2 215.1812} C_DIS
LIN {X -77.8425,Y -114.7826,Z 162,A -126.749,B 24.97,C -1.2658,E1 24.9113,E2 213.4469} C_DIS
LIN {X -74.3011,Y -117.1065,Z 162,A -124.9101,B 24.97,C -1.2677,E1 24.9156,E2 211.5974} C_DIS
LIN {X -70.3535,Y -119.5193,Z 162,A -123.0142,B 24.97,C -1.264,E1 24.9201,E2 209.7045} C_DIS
LIN {X -66.3593,Y -121.7823,Z 162,A -121.0791,B 24.9701,C -1.2634,E1 24.9249,E2 207.7653} C_DIS
LIN {X -62.7156,Y -123.6961,Z 162,A -119.4554,B 24.9704,C -1.257,E1 24.9289,E2 206.1522} C_DIS
LIN {X -60.2537,Y -124.9147,Z 162,A -117.8745,B 24.9693,C -1.2798,E1 24.933,E2 204.5132} C_DIS
LIN {X -56.3041,Y -126.7434,Z 162,A -116.4433,B 24.9704,C -1.2578,E1 24.9365,E2 203.1308} C_DIS
LIN {X -52.6601,Y -128.3027,Z 162,A -114.7859,B 24.9704,C -1.2571,E1 24.9408,E2 201.4714} C_DIS
LIN {X -49.2756,Y -129.6392,Z 162,A -113.3327,B 24.9706,C -1.2529,E1 24.9446,E2 200.025} C_DIS
LIN {X -45.8448,Y -130.8908,Z 162,A -111.9392,B 24.971,C -1.2453,E1 24.9482,E2 198.6468} C_DIS
LIN {X -42.7621,Y -131.9307,Z 162,A -110.5853,B 24.971,C -1.2447,E1 24.9518,E2 197.2918} C_DIS
LIN {X -39.6107,Y -132.9113,Z 162,A -109.2142,B 24.971,C -1.2441,E1 24.9555,E2 195.9198} C_DIS
LIN {X -36.5306,Y -133.7915,Z 162,A -107.8735,B 24.971,C -1.2441,E1 24.9591,E2 194.5769} C_DIS
LIN {X -33.3247,Y -134.6259,Z 162,A -106.3552,B 24.9707,C -1.2515,E1 24.9632,E2 193.0388} C_DIS
LIN {X -27.1465,Y -136.0049,Z 162,A -103.7476,B 24.9707,C -1.2499,E1 24.9704,E2 190.432} C_DIS
LIN {X -22.9492,Y -136.7749,Z 162,A -102.0959,B 24.9711,C -1.2432,E1 24.9749,E2 188.7945} C_DIS
LIN {X -18.9711,Y -137.3847,Z 162,A -100.4927,B 24.9712,C -1.2394,E1 24.9793,E2 187.1989} C_DIS
LIN {X -15.9758,Y -137.7644,Z 162,A -99.0765,B 24.9708,C -1.2486,E1 24.9833,E2 185.7601} C_DIS
LIN {X -11.9251,Y -138.1735,Z 162,A -97.445,B 24.9709,C -1.2457,E1 24.9878,E2 184.1347} C_DIS
LIN {X -7.7419,Y -138.4728,Z 162,A -95.6797,B 24.9709,C -1.2475,E1 24.9927,E2 182.3644} C_DIS
LIN {X -4.3516,Y -138.6196,Z 162,A -94.415,B 24.9712,C -1.24,E1 24.9962,E2 181.1172} C_DIS
LIN {X -0.49,Y -138.6864,Z 162,A -92.7121,B 24.9709,C -1.2463,E1 25.001,E2 179.3993} C_DIS
LIN {X -0.49,Y -138.6864,Z 162,A -92.7121,B 24.9709,C -1.2463,E1 25.001,E2 179.3993} C_DIS
Enddeposition()
LIN {X 0.973,Y -137.7564,Z 162,A -92.7661,B 24.9718,C -1.2263,E1 25.0007,E2 179.5007} C_DIS
Startdeposition()
$VEL.CP = VEL_PRINT
LIN {X -5.0168,Y -137.6733,Z 162,A -95.4088,B 24.9722,C -1.2176,E1 24.9933,E2 182.1643} C_DIS
LIN {X -9.0549,Y -137.4675,Z 162,A -97.021,B 24.9721,C -1.2213,E1 24.9888,E2 183.7683} C_DIS
LIN {X -13.8579,Y -137.0662,Z 162,A -99.6342,B 24.9735,C -1.1887,E1 24.9813,E2 186.4602} C_DIS
LIN {X -18.8833,Y -136.4651,Z 162,A -101.0363,B 24.9718,C -1.2269,E1 24.9777,E2 187.7727} C_DIS
LIN {X -27.0562,Y -135.0816,Z 162,A -104.8623,B 24.9727,C -1.2077,E1 24.967,E2 191.6481} C_DIS
LIN {X -30.2453,Y -134.4036,Z 162,A -105.9339,B 24.972,C -1.2236,E1 24.9642,E2 192.6834} C_DIS
LIN {X -33.4884,Y -133.6323,Z 162,A -107.356,B 24.972,C -1.2224,E1 24.9603,E2 194.1101} C_DIS
LIN {X -36.9051,Y -132.7288,Z 162,A -108.7974,B 24.972,C -1.2249,E1 24.9565,E2 195.5478} C_DIS
LIN {X -40.295,Y -131.7391,Z 162,A -110.2599,B 24.9718,C -1.2263,E1 24.9525,E2 197.0095} C_DIS
LIN {X -43.361,Y -130.7621,Z 162,A -111.6173,B 24.9718,C -1.2263,E1 24.9489,E2 198.3692} C_DIS
LIN {X -46.672,Y -129.6171,Z 162,A -113.155,B 24.972,C -1.2234,E1 24.9449,E2 199.917} C_DIS
LIN {X -50.8091,Y -128.0541,Z 162,A -114.9536,B 24.9718,C -1.2273,E1 24.9402,E2 201.71} C_DIS
LIN {X -53.8847,Y -126.7909,Z 162,A -116.4991,B 24.9721,C -1.2202,E1 24.9362,E2 203.2761} C_DIS
LIN {X -58.0707,Y -124.9268,Z 162,A -118.3257,B 24.9718,C -1.2266,E1 24.9315,E2 205.0919} C_DIS
LIN {X -62.0632,Y -122.9928,Z 162,A -120.096,B 24.9715,C -1.2329,E1 24.9271,E2 206.8519} C_DIS
LIN {X -65.463,Y -121.2191,Z 162,A -121.7711,B 24.9716,C -1.2308,E1 24.923,E2 208.5367} C_DIS
LIN {X -69.4894,Y -118.9568,Z 162,A -123.703,B 24.9716,C -1.233,E1 24.9183,E2 210.469} C_DIS
LIN {X -73.3018,Y -116.6461,Z 162,A -125.5597,B 24.9714,C -1.2358,E1 24.9139,E2 212.325} C_DIS
LIN {X -77.1809,Y -114.1161,Z 162,A -127.4385,B 24.9711,C -1.2414,E1 24.9095,E2 214.1966} C_DIS
LIN {X -80.734,Y -111.6307,Z 162,A -128.97,B 24.9703,C -1.2588,E1 24.9061,E2 215.6921} C_DIS
LIN {X -83.6698,Y -109.4474,Z 162,A -130.8144,B 24.971,C -1.2446,E1 24.9019,E2 217.5767} C_DIS
LIN {X -87.5173,Y -106.3968,Z 162,A -133.5748,B 24.9725,C -1.2115,E1 24.8958,E2 220.4263} C_DIS
LIN {X -92.1255,Y -102.4321,Z 162,A -135.3816,B 24.9706,C -1.2537,E1 24.8922,E2 222.1398} C_DIS
LIN {X -95.5549,Y -99.241,Z 162,A -137.3129,B 24.9703,C -1.2587,E1 24.8883,E2 224.0671} C_DIS
LIN {X -98.6919,Y -96.122,Z 162,A -139.2086,B 24.9703,C -1.2599,E1 24.8845,E2 225.9682} C_DIS
LIN {X -101.7878,Y -92.8372,Z 162,A -141.1271,B 24.9702,C -1.2621,E1 24.8809,E2 227.89} C_DIS
LIN {X -105.4147,Y -88.697,Z 162,A -143.3811,B 24.9698,C -1.2693,E1 24.8768,E2 230.1369} C_DIS
LIN {X -108.081,Y -85.4287,Z 162,A -145.1972,B 24.9698,C -1.2704,E1 24.8736,E2 231.9589} C_DIS
LIN {X -111.148,Y -81.3974,Z 162,A -147.1425,B 24.9691,C -1.284,E1 24.8704,E2 233.8812} C_DIS
LIN {X -115.3064,Y -75.3923,Z 162,A -150.3645,B 24.9691,C -1.2825,E1 24.8653,E2 237.1227} C_DIS
LIN {X -117.6702,Y -71.6469,Z 162,A -152.2131,B 24.969,C -1.2872,E1 24.8626,E2 238.9698} C_DIS
LIN {X -119.7649,Y -68.0866,Z 162,A -153.9332,B 24.9687,C -1.2918,E1 24.8602,E2 240.6878} C_DIS
LIN {X -121.7738,Y -64.4215,Z 162,A -155.5893,B 24.9683,C -1.3009,E1 24.858,E2 242.3309} C_DIS
LIN {X -123.5211,Y -61.0031,Z 162,A -157.8958,B 24.9698,C -1.2697,E1 24.855,E2 244.7243} C_DIS
LIN {X -125.9297,Y -55.8635,Z 162,A -159.6009,B 24.9679,C -1.3096,E1 24.8532,E2 246.3437} C_DIS
LIN {X -127.6446,Y -51.8249,Z 162,A -161.3838,B 24.9675,C -1.3172,E1 24.8512,E2 248.1184} C_DIS
LIN {X -129.0251,Y -48.2843,Z 162,A -163.0157,B 24.9674,C -1.3193,E1 24.8496,E2 249.7543} C_DIS
LIN {X -130.4273,Y -44.3648,Z 162,A -165.4132,B 24.9688,C -1.2912,E1 24.8474,E2 252.2326} C_DIS
LIN {X -132.0715,Y -39.1952,Z 162,A -167.1862,B 24.9672,C -1.3224,E1 24.846,E2 253.9414} C_DIS
LIN {X -133.3178,Y -34.7259,Z 162,A -169.0589,B 24.9668,C -1.3313,E1 24.8446,E2 255.8037} C_DIS
LIN {X -134.278,Y -30.7951,Z 162,A -170.6334,B 24.9663,C -1.3421,E1 24.8436,E2 257.3617} C_DIS
LIN {X -135.011,Y -27.4034,Z 162,A -172.1357,B 24.9662,C -1.3438,E1 24.8428,E2 258.8689} C_DIS
LIN {X -135.8036,Y -23.1636,Z 162,A -173.8872,B 24.9658,C -1.3517,E1 24.8419,E2 260.6119} C_DIS
LIN {X -136.3449,Y -19.7248,Z 162,A -175.3479,B 24.9656,C -1.3558,E1 24.8413,E2 262.0717} C_DIS
LIN {X -136.7976,Y -16.2902,Z 162,A -176.7839,B 24.9653,C -1.3607,E1 24.8408,E2 263.5045} C_DIS
LIN {X -137.2197,Y -12.2537,Z 162,A -178.6016,B 24.9653,C -1.3597,E1 24.8403,E2 265.3354} C_DIS
LIN {X -137.5067,Y -8.4189,Z 162,A 179.8945,B 24.9649,C -1.3698,E1 24.84,E2 266.8243} C_DIS
LIN {X -137.6996,Y -4.2415,Z 162,A 178.085,B 24.9647,C -1.372,E1 24.8398,E2 268.6395} C_DIS
LIN {X -137.767,Y -0.1145,Z 162,A 176.443,B 24.9643,C -1.3814,E1 24.8398,E2 270.2689} C_DIS
LIN {X -137.7385,Y 2.6935,Z 162,A 175.2467,B 24.9641,C -1.3839,E1 24.8398,E2 271.4665} C_DIS
LIN {X -137.6172,Y 6.3825,Z 162,A 173.5632,B 24.9642,C -1.3816,E1 24.84,E2 273.1657} C_DIS
LIN {X -137.3423,Y 10.8002,Z 162,A 171.7172,B 24.9639,C -1.3874,E1 24.8404,E2 275.0089} C_DIS
LIN {X -136.9772,Y 14.7033,Z 162,A 170.1537,B 24.9635,C -1.3962,E1 24.8408,E2 276.5608} C_DIS
LIN {X -136.4317,Y 19.1174,Z 162,A 168.291,B 24.9632,C -1.4017,E1 24.8415,E2 278.4215} C_DIS
LIN {X -135.8726,Y 22.75,Z 162,A 166.7732,B 24.9629,C -1.4073,E1 24.8422,E2 279.935} C_DIS
LIN {X -135.0972,Y 26.9799,Z 162,A 164.9314,B 24.9627,C -1.4105,E1 24.8431,E2 281.7801} C_DIS
LIN {X -134.36,Y 30.436,Z 162,A 163.5047,B 24.9624,C -1.4175,E1 24.844,E2 283.1985} C_DIS
LIN {X -133.5387,Y 33.8572,Z 162,A 162.0368,B 24.9621,C -1.4221,E1 24.845,E2 284.6641} C_DIS
LIN {X -132.6057,Y 37.3455,Z 162,A 160.525,B 24.9619,C -1.4264,E1 24.8461,E2 286.1743} C_DIS
LIN {X -131.5424,Y 40.9377,Z 162,A 158.8518,B 24.9619,C -1.4257,E1 24.8475,E2 287.8589} C_DIS
LIN {X -130.275,Y 44.804,Z 162,A 157.2508,B 24.9614,C -1.4357,E1 24.8489,E2 289.4451} C_DIS
LIN {X -129.1022,Y 48.0785,Z 162,A 155.6374,B 24.9616,C -1.432,E1 24.8504,E2 291.0766} C_DIS
LIN {X -126.7829,Y 53.9038,Z 162,A 153.0358,B 24.9611,C -1.4405,E1 24.8532,E2 293.6724} C_DIS
LIN {X -125.2344,Y 57.4054,Z 162,A 151.6051,B 24.9604,C -1.4535,E1 24.8548,E2 295.0798} C_DIS
LIN {X -123.8993,Y 60.2364,Z 162,A 150.1803,B 24.9605,C -1.4514,E1 24.8565,E2 296.5176} C_DIS
LIN {X -122.1961,Y 63.6174,Z 162,A 148.6991,B 24.96,C -1.4609,E1 24.8584,E2 297.984} C_DIS
LIN {X -120.8741,Y 66.0973,Z 162,A 147.2177,B 24.9607,C -1.4487,E1 24.8604,E2 299.5023} C_DIS
LIN {X -119.2694,Y 68.9507,Z 162,A 146.0471,B 24.9599,C -1.4623,E1 24.862,E2 300.6465} C_DIS
LIN {X -117.6032,Y 71.7563,Z 162,A 144.7095,B 24.9597,C -1.4672,E1 24.8639,E2 301.9792} C_DIS
LIN {X -115.4221,Y 75.2141,Z 162,A 142.3954,B 24.9611,C -1.4414,E1 24.8676,E2 304.3665} C_DIS
LIN {X -112.4438,Y 79.5979,Z 162,A 140.7912,B 24.9591,C -1.4777,E1 24.87,E2 305.8922} C_DIS
LIN {X -109.8319,Y 83.1648,Z 162,A 138.9355,B 24.9589,C -1.482,E1 24.8731,E2 307.7467} C_DIS
LIN {X -107.1822,Y 86.5527,Z 162,A 136.8145,B 24.9595,C -1.4701,E1 24.8769,E2 309.9058} C_DIS
LIN {X -104.7603,Y 89.4693,Z 162,A 135.5136,B 24.9585,C -1.4882,E1 24.8791,E2 311.1696} C_DIS
LIN {X -101.8733,Y 92.7429,Z 162,A 133.7034,B 24.9582,C -1.4932,E1 24.8825,E2 312.9761} C_DIS
LIN {X -98.8826,Y 95.925,Z 162,A 131.8756,B 24.958,C -1.4972,E1 24.886,E2 314.8022} C_DIS
LIN {X -95.6092,Y 99.1884,Z 162,A 129.9578,B 24.9577,C -1.5022,E1 24.8898,E2 316.7162} C_DIS
LIN {X -92.4905,Y 102.1024,Z 162,A 128.1702,B 24.9575,C -1.5058,E1 24.8935,E2 318.5024} C_DIS
LIN {X -89.1788,Y 105.0072,Z 162,A 126.3178,B 24.9573,C -1.509,E1 24.8974,E2 320.3544} C_DIS
LIN {X -85.7988,Y 107.7865,Z 162,A 124.5528,B 24.9569,C -1.5159,E1 24.9012,E2 322.1097} C_DIS
LIN {X -82.6482,Y 110.2217,Z 162,A 122.8058,B 24.957,C -1.5148,E1 24.9051,E2 323.8656} C_DIS
LIN {X -79.0569,Y 112.8254,Z 162,A 120.9232,B 24.9569,C -1.5168,E1 24.9094,E2 325.75} C_DIS
LIN {X -75.255,Y 115.3952,Z 162,A 118.7159,B 24.9575,C -1.5053,E1 24.9146,E2 327.9918} C_DIS
LIN {X -71.8668,Y 117.5354,Z 162,A 117.4651,B 24.9562,C -1.5298,E1 24.9175,E2 329.1884} C_DIS
LIN {X -63.4045,Y 122.3079,Z 162,A 113.3454,B 24.956,C -1.5329,E1 24.9276,E2 333.3127} C_DIS
LIN {X -59.783,Y 124.117,Z 162,A 111.7165,B 24.9557,C -1.5385,E1 24.9316,E2 334.9325} C_DIS
LIN {X -56.5226,Y 125.6349,Z 162,A 110.1876,B 24.9557,C -1.5391,E1 24.9355,E2 336.4637} C_DIS
LIN {X -53.3479,Y 127.0155,Z 162,A 108.4143,B 24.9565,C -1.524,E1 24.9402,E2 338.277} C_DIS
LIN {X -49.9741,Y 128.3801,Z 162,A 107.0786,B 24.9558,C -1.5353,E1 24.9436,E2 339.5888} C_DIS
LIN {X -45.5129,Y 130.0293,Z 162,A 105.2369,B 24.9553,C -1.5449,E1 24.9484,E2 341.4112} C_DIS
LIN {X -42.1871,Y 131.1457,Z 162,A 103.7419,B 24.9553,C -1.5449,E1 24.9523,E2 342.9091} C_DIS
LIN {X -36.341,Y 132.8866,Z 162,A 101.1512,B 24.9553,C -1.5449,E1 24.9593,E2 345.5041} C_DIS
LIN {X -32.5733,Y 133.858,Z 162,A 99.6477,B 24.9548,C -1.5525,E1 24.9633,E2 346.9916} C_DIS
LIN {X -29.1794,Y 134.6383,Z 162,A 98.1882,B 24.9548,C -1.5532,E1 24.9673,E2 348.4512} C_DIS
LIN {X -25.866,Y 135.314,Z 162,A 96.774,B 24.9548,C -1.554,E1 24.9712,E2 349.8651} C_DIS
LIN {X -22.1576,Y 135.9715,Z 162,A 95.1051,B 24.955,C -1.5498,E1 24.9758,E2 351.5458} C_DIS
LIN {X -17.8518,Y 136.6025,Z 162,A 92.9859,B 24.9559,C -1.5347,E1 24.9818,E2 353.7023} C_DIS
LIN {X -13.8056,Y 137.0721,Z 162,A 91.4509,B 24.9553,C -1.5439,E1 24.986,E2 355.2162} C_DIS
LIN {X -9.4665,Y 137.4397,Z 162,A 89.218,B 24.9566,C -1.5225,E1 24.9924,E2 357.5007} C_DIS
LIN {X -4.1369,Y 137.7025,Z 162,A 87.8758,B 24.9538,C -1.5696,E1 24.9958,E2 358.7316} C_DIS
LIN {X 2.6134,Y 137.7398,Z 162,A 84.9265,B 24.9543,C -1.5625,E1 25.0041,E2 361.6976} C_DIS
LIN {X 8.5352,Y 137.4995,Z 162,A 82.7397,B 24.9534,C -1.5775,E1 25.0101,E2 363.8482} C_DIS
LIN {X 15.2778,Y 136.9154,Z 162,A 79.6069,B 24.9544,C -1.56,E1 25.0189,E2 367.0206} C_DIS
LIN {X 19.4554,Y 136.3834,Z 162,A 77.2998,B 24.9562,C -1.5299,E1 25.0255,E2 369.3972} C_DIS
LIN {X 24.0224,Y 135.6536,Z 162,A 75.7248,B 24.9551,C -1.5478,E1 25.0297,E2 370.9281} C_DIS
LIN {X 28.8252,Y 134.7148,Z 162,A 73.805,B 24.9548,C -1.553,E1 25.0349,E2 372.8331} C_DIS
LIN {X 32.8834,Y 133.7833,Z 162,A 72.0127,B 24.9551,C -1.5487,E1 25.0398,E2 374.633} C_DIS
LIN {X 36.9294,Y 132.722,Z 162,A 70.4195,B 24.9547,C -1.5555,E1 25.044,E2 376.2076} C_DIS
LIN {X 40.2377,Y 131.7566,Z 162,A 68.9711,B 24.9547,C -1.5536,E1 25.0479,E2 377.658} C_DIS
LIN {X 43.4063,Y 130.747,Z 162,A 67.5034,B 24.9551,C -1.5479,E1 25.0518,E2 379.1365} C_DIS
LIN {X 47.9186,Y 129.1621,Z 162,A 65.6406,B 24.9548,C -1.5529,E1 25.0567,E2 380.9837} C_DIS
LIN {X 51.4147,Y 127.81,Z 162,A 63.9551,B 24.9553,C -1.5444,E1 25.0611,E2 382.6856} C_DIS
LIN {X 55.1152,Y 126.2592,Z 162,A 62.2658,B 24.9555,C -1.5413,E1 25.0654,E2 384.378} C_DIS
LIN {X 59.0027,Y 124.4897,Z 162,A 60.5977,B 24.9553,C -1.5451,E1 25.0696,E2 386.0329} C_DIS
LIN {X 62.2447,Y 122.9004,Z 162,A 59.156,B 24.9552,C -1.5465,E1 25.0732,E2 387.4676} C_DIS
LIN {X 65.5556,Y 121.1693,Z 162,A 57.4827,B 24.9557,C -1.5377,E1 25.0774,E2 389.1568} C_DIS
LIN {X 69.3389,Y 119.0446,Z 162,A 55.6582,B 24.9559,C -1.5339,E1 25.0818,E2 390.9847} C_DIS
LIN {X 73.189,Y 116.7172,Z 162,A 53.781,B 24.9561,C -1.5306,E1 25.0863,E2 392.8638} C_DIS
LIN {X 77.0482,Y 114.2059,Z 162,A 52.0136,B 24.9558,C -1.5356,E1 25.0903,E2 394.6136} C_DIS
LIN {X 80.2236,Y 111.998,Z 162,A 50.3424,B 24.9562,C -1.5293,E1 25.0942,E2 396.2938} C_DIS
LIN {X 83.6856,Y 109.4353,Z 162,A 48.5734,B 24.9562,C -1.5273,E1 25.0981,E2 398.0612} C_DIS
LIN {X 86.8754,Y 106.9214,Z 162,A 46.4458,B 24.9579,C -1.4997,E1 25.1029,E2 400.246} C_DIS
LIN {X 90.2301,Y 104.1061,Z 162,A 44.993,B 24.9569,C -1.5165,E1 25.1059,E2 401.6535} C_DIS
LIN {X 93.4884,Y 101.19,Z 162,A 43.2062,B 24.957,C -1.5145,E1 25.1095,E2 403.4378} C_DIS
LIN {X 96.8963,Y 97.9314,Z 162,A 41.2332,B 24.9573,C -1.5095,E1 25.1135,E2 405.4142} C_DIS
LIN {X 99.9858,Y 94.7751,Z 162,A 39.4296,B 24.9574,C -1.5073,E1 25.117,E2 407.2154} C_DIS
LIN {X 102.2576,Y 92.3194,Z 162,A 37.9962,B 24.9578,C -1.5017,E1 25.1197,E2 408.6557} C_DIS
LIN {X 105.3288,Y 88.7993,Z 162,A 36.0949,B 24.9578,C -1.4994,E1 25.1231,E2 410.5538} C_DIS
LIN {X 108.1658,Y 85.3206,Z 162,A 34.2387,B 24.9581,C -1.4954,E1 25.1264,E2 412.4108} C_DIS
LIN {X 110.9793,Y 81.6271,Z 162,A 32.3915,B 24.9581,C -1.4952,E1 25.1295,E2 414.2496} C_DIS
LIN {X 113.9697,Y 77.3972,Z 162,A 30.1788,B 24.9586,C -1.4863,E1 25.133,E2 416.4724} C_DIS
LIN {X 116.4776,Y 73.5687,Z 162,A 28.326,B 24.9587,C -1.484,E1 25.1358,E2 418.3213} C_DIS
LIN {X 118.7799,Y 69.7906,Z 162,A 26.5005,B 24.959,C -1.4798,E1 25.1384,E2 420.1474} C_DIS
LIN {X 120.8811,Y 66.0845,Z 162,A 24.756,B 24.9592,C -1.4764,E1 25.1408,E2 421.8908} C_DIS
LIN {X 122.5851,Y 62.864,Z 162,A 23.2933,B 24.9592,C -1.4751,E1 25.1427,E2 423.3488} C_DIS
LIN {X 124.1615,Y 59.6897,Z 162,A 21.8676,B 24.9593,C -1.4736,E1 25.1444,E2 424.7704} C_DIS
LIN {X 125.6139,Y 56.5695,Z 162,A 20.4219,B 24.9596,C -1.4685,E1 25.1461,E2 426.2203} C_DIS
LIN {X 126.9262,Y 53.5615,Z 162,A 19.044,B 24.9599,C -1.4637,E1 25.1476,E2 427.6019} C_DIS
LIN {X 128.3344,Y 50.0916,Z 162,A 17.5826,B 24.9599,C -1.4646,E1 25.1492,E2 429.0533} C_DIS
LIN {X 129.5071,Y 46.977,Z 162,A 16.1979,B 24.9601,C -1.4603,E1 25.1505,E2 430.4403} C_DIS
LIN {X 130.6592,Y 43.67,Z 162,A 14.1079,B 24.9622,C -1.4197,E1 25.1524,E2 432.6141} C_DIS
LIN {X 132.1257,Y 39.0101,Z 162,A 12.6738,B 24.9608,C -1.4474,E1 25.1535,E2 433.9748} C_DIS
LIN {X 133.1164,Y 35.4813,Z 162,A 11.1483,B 24.961,C -1.4425,E1 25.1547,E2 435.5031} C_DIS
LIN {X 133.9161,Y 32.3323,Z 162,A 9.7773,B 24.9613,C -1.4371,E1 25.1556,E2 436.8789} C_DIS
LIN {X 134.8223,Y 28.3275,Z 162,A 7.9711,B 24.9619,C -1.4259,E1 25.1567,E2 438.7009} C_DIS
LIN {X 135.5512,Y 24.5945,Z 162,A 6.5359,B 24.9617,C -1.4293,E1 25.1574,E2 440.1198} C_DIS
LIN {X 136.3637,Y 19.5934,Z 162,A 4.3143,B 24.9624,C -1.4159,E1 25.1584,E2 442.36} C_DIS
LIN {X 136.8643,Y 15.7312,Z 162,A 2.2742,B 24.964,C -1.3865,E1 25.1591,E2 444.4572} C_DIS
LIN {X 137.3326,Y 10.9169,Z 162,A 0.9563,B 24.9623,C -1.4196,E1 25.1593,E2 445.6894} C_DIS
LIN {X 137.6914,Y 4.5348,Z 162,A -1.8926,B 24.9633,C -1.3997,E1 25.1598,E2 448.568} C_DIS
LIN {X 137.7509,Y -1.951,Z 162,A -4.2869,B 24.9629,C -1.4083,E1 25.1598,E2 450.928} C_DIS
LIN {X 137.6574,Y -5.4243,Z 162,A -6.2001,B 24.9645,C -1.3765,E1 25.1596,E2 452.9047} C_DIS
LIN {X 137.4875,Y -8.731,Z 162,A -6.9902,B 24.963,C -1.4057,E1 25.1595,E2 453.6212} C_DIS
LIN {X 136.9339,Y -15.1064,Z 162,A -9.8499,B 24.9641,C -1.3853,E1 25.1588,E2 456.5121} C_DIS
LIN {X 136.0266,Y -21.8236,Z 162,A -12.8719,B 24.9651,C -1.3642,E1 25.1576,E2 459.5661} C_DIS
LIN {X 135.3876,Y -25.4806,Z 162,A -14.3696,B 24.9653,C -1.3617,E1 25.1568,E2 461.0608} C_DIS
LIN {X 134.5934,Y -29.3873,Z 162,A -16.0157,B 24.9655,C -1.3569,E1 25.1558,E2 462.7086} C_DIS
LIN {X 133.4149,Y -34.3449,Z 162,A -18.1299,B 24.9658,C -1.3503,E1 25.1544,E2 464.8262} C_DIS
LIN {X 132.3368,Y -38.289,Z 162,A -19.6673,B 24.9657,C -1.3541,E1 25.1533,E2 466.3458} C_DIS
LIN {X 131.2873,Y -41.7438,Z 162,A -21.1459,B 24.9658,C -1.3506,E1 25.1521,E2 467.8243} C_DIS
LIN {X 130.1776,Y -45.085,Z 162,A -22.5985,B 24.966,C -1.3465,E1 25.1508,E2 469.2782} C_DIS
LIN {X 129.1552,Y -47.9371,Z 162,A -24.2412,B 24.9673,C -1.3205,E1 25.1491,E2 470.9731} C_DIS
LIN {X 127.8635,Y -51.2819,Z 162,A -25.2158,B 24.9661,C -1.3455,E1 25.1482,E2 471.8835} C_DIS
LIN {X 125.5216,Y -56.7759,Z 162,A -27.9734,B 24.9673,C -1.3218,E1 25.1451,E2 474.6816} C_DIS
LIN {X 123.7505,Y -60.538,Z 162,A -29.5971,B 24.9673,C -1.3226,E1 25.1431,E2 476.2949} C_DIS
LIN {X 121.7696,Y -64.4296,Z 162,A -31.3894,B 24.9674,C -1.3184,E1 25.1408,E2 478.0876} C_DIS
LIN {X 119.8423,Y -67.951,Z 162,A -33.148,B 24.9679,C -1.3082,E1 25.1384,E2 479.861} C_DIS
LIN {X 117.6725,Y -71.6431,Z 162,A -34.8553,B 24.9679,C -1.3071,E1 25.136,E2 481.5621} C_DIS
LIN {X 115.7444,Y -74.7178,Z 162,A -36.3653,B 24.9682,C -1.3027,E1 25.1337,E2 483.0751} C_DIS
LIN {X 112.6064,Y -79.3674,Z 162,A -38.6967,B 24.9685,C -1.2961,E1 25.13,E2 485.4105} C_DIS
LIN {X 109.9141,Y -83.0558,Z 162,A -40.5927,B 24.9688,C -1.2909,E1 25.1269,E2 487.3096} C_DIS
LIN {X 107.0254,Y -86.7471,Z 162,A -42.5353,B 24.969,C -1.2859,E1 25.1235,E2 489.2548} C_DIS
LIN {X 104.0975,Y -90.2401,Z 162,A -44.436,B 24.9693,C -1.2806,E1 25.12,E2 491.1595} C_DIS
LIN {X 101.2022,Y -93.4751,Z 162,A -46.2267,B 24.9695,C -1.2767,E1 25.1167,E2 492.9514} C_DIS
LIN {X 98.1286,Y -96.6967,Z 162,A -48.0357,B 24.9695,C -1.2744,E1 25.1132,E2 494.7581} C_DIS
LIN {X 95.0085,Y -99.7638,Z 162,A -49.8521,B 24.9698,C -1.2701,E1 25.1095,E2 496.5771} C_DIS
LIN {X 91.6928,Y -102.8197,Z 162,A -51.7455,B 24.9701,C -1.2645,E1 25.1056,E2 498.4759} C_DIS
LIN {X 88.2649,Y -105.7772,Z 162,A -53.6284,B 24.9703,C -1.2601,E1 25.1016,E2 500.3618} C_DIS
LIN {X 84.7084,Y -108.6463,Z 162,A -55.5352,B 24.9705,C -1.2555,E1 25.0974,E2 502.2725} C_DIS
LIN {X 81.0959,Y -111.3684,Z 162,A -57.3874,B 24.9705,C -1.2531,E1 25.0932,E2 504.1239} C_DIS
LIN {X 77.4925,Y -113.9052,Z 162,A -59.2306,B 24.9708,C -1.2487,E1 25.089,E2 505.9711} C_DIS
LIN {X 73.6102,Y -116.4514,Z 162,A -61.0999,B 24.9708,C -1.2483,E1 25.0846,E2 507.8353} C_DIS
LIN {X 69.9275,Y -118.6994,Z 162,A -62.8868,B 24.971,C -1.2453,E1 25.0803,E2 509.6237} C_DIS
LIN {X 66.1758,Y -120.8313,Z 162,A -64.6063,B 24.971,C -1.2462,E1 25.0762,E2 511.3359} C_DIS
LIN {X 62.8058,Y -122.6147,Z 162,A -66.5804,B 24.972,C -1.2218,E1 25.0711,E2 513.3623} C_DIS
LIN {X 59.3356,Y -124.3307,Z 162,A -67.7353,B 24.971,C -1.2446,E1 25.0684,E2 514.4603} C_DIS
LIN {X 56.4869,Y -125.6508,Z 162,A -69.4056,B 24.972,C -1.2221,E1 25.064,E2 516.1795} C_DIS
LIN {X 53.315,Y -127.0292,Z 162,A -70.5089,B 24.9713,C -1.2386,E1 25.0613,E2 517.2412} C_DIS
LIN {X 50.2308,Y -128.2803,Z 162,A -72.4274,B 24.9727,C -1.2069,E1 25.0561,E2 519.2303} C_DIS
LIN {X 45.8372,Y -129.9168,Z 162,A -73.8478,B 24.9715,C -1.2336,E1 25.0526,E2 520.5847} C_DIS
LIN {X 42.0112,Y -131.2019,Z 162,A -75.5293,B 24.9716,C -1.2314,E1 25.0481,E2 522.2683} C_DIS
LIN {X 38.2638,Y -132.3442,Z 162,A -77.1982,B 24.9718,C -1.2273,E1 25.0436,E2 523.9441} C_DIS
LIN {X 34.0714,Y -133.4843,Z 162,A -78.8937,B 24.9716,C -1.2315,E1 25.0391,E2 525.6268} C_DIS
LIN {X 30.7584,Y -134.2864,Z 162,A -80.3652,B 24.9718,C -1.2271,E1 25.035,E2 527.1066} C_DIS
LIN {X 27.2614,Y -135.0399,Z 162,A -82.1875,B 24.9727,C -1.2073,E1 25.0299,E2 528.9735} C_DIS
LIN {X 23.7036,Y -135.7102,Z 162,A -83.4655,B 24.9722,C -1.2186,E1 25.0265,E2 530.2234} C_DIS
LIN {X 20.3562,Y -136.2538,Z 162,A -84.915,B 24.9723,C -1.2154,E1 25.0225,E2 531.6791} C_DIS
LIN {X 14.9215,Y -136.9538,Z 162,A -86.8798,B 24.9716,C -1.2312,E1 25.0171,E2 533.6049} C_DIS
LIN {X 7.9868,Y -137.5333,Z 162,A -90.047,B 24.9724,C -1.2148,E1 25.0082,E2 536.8095} C_DIS
LIN {X 3.879,Y -137.7096,Z 162,A -91.6862,B 24.9722,C -1.2181,E1 25.0037,E2 538.4406} C_DIS
LIN {X 0.973,Y -137.7564,Z 162,A -92.763,B 24.9719,C -1.225,E1 25.0007,E2 539.5007} C_DIS
Enddeposition()
LIN {X 0.973,Y -137.7564,Z 162,A -92.763,B 24.9719,C -1.225,E1 25.0007,E2 539.5007} C_DIS
Startdeposition()
$VEL.CP = VEL_PRINT
LIN {X 4.2002,Y -136.7776,Z 162,A -89.7788,B 22.5482,C -0.8462,E1 22.5704,E2 537.169} C_DIS
LIN {X 7.4345,Y -136.6405,Z 162,A -88.8254,B 22.5489,C -0.8267,E1 22.5729,E2 536.2666} C_DIS
LIN {X 13.7917,Y -136.1464,Z 162,A -85.6482,B 22.548,C -0.8532,E1 22.582,E2 533.0224} C_DIS
LIN {X 17.4425,Y -135.7255,Z 162,A -84.425,B 22.5485,C -0.8384,E1 22.5852,E2 531.8388} C_DIS
LIN {X 21.482,Y -135.1457,Z 162,A -82.731,B 22.5485,C -0.8389,E1 22.5899,E2 530.1455} C_DIS
LIN {X 27.0561,Y -134.14,Z 162,A -80.385,B 22.5485,C -0.8395,E1 22.5963,E2 527.8008} C_DIS
LIN {X 30.9135,Y -133.3044,Z 162,A -78.6552,B 22.5482,C -0.8449,E1 22.6011,E2 526.0597} C_DIS
LIN {X 35.0845,Y -132.2672,Z 162,A -77.031,B 22.5485,C -0.8379,E1 22.6054,E2 524.4564} C_DIS
LIN {X 38.5768,Y -131.291,Z 162,A -75.4405,B 22.5483,C -0.8432,E1 22.6097,E2 522.8551} C_DIS
LIN {X 42.364,Y -130.1205,Z 162,A -73.7444,B 22.5482,C -0.847,E1 22.6142,E2 521.1528} C_DIS
LIN {X 45.2884,Y -129.1304,Z 162,A -71.773,B 22.5469,C -0.8832,E1 22.6197,E2 519.0916} C_DIS
LIN {X 50.6709,Y -127.1149,Z 162,A -70.2406,B 22.5484,C -0.8419,E1 22.6234,E2 517.6703} C_DIS
LIN {X 55.3878,Y -125.1316,Z 162,A -67.9018,B 22.5479,C -0.855,E1 22.6295,E2 515.3037} C_DIS
LIN {X 58.8794,Y -123.526,Z 162,A -66.5759,B 22.5483,C -0.8432,E1 22.6327,E2 514.0124} C_DIS
LIN {X 61.0791,Y -122.4546,Z 162,A -65.0722,B 22.5474,C -0.8692,E1 22.6366,E2 512.4456} C_DIS
LIN {X 65.5272,Y -120.1339,Z 162,A -63.2015,B 22.5477,C -0.861,E1 22.6412,E2 510.6021} C_DIS
LIN {X 69.3385,Y -117.9752,Z 162,A -61.4071,B 22.5477,C -0.8623,E1 22.6455,E2 508.8104} C_DIS
LIN {X 72.8991,Y -115.809,Z 162,A -59.6201,B 22.5474,C -0.8678,E1 22.6498,E2 507.0156} C_DIS
LIN {X 76.6093,Y -113.3887,Z 162,A -57.7806,B 22.5474,C -0.8706,E1 22.654,E2 505.1756} C_DIS
LIN {X 80.1729,Y -110.8977,Z 162,A -55.949,B 22.5472,C -0.8749,E1 22.6582,E2 503.34} C_DIS
LIN {X 83.7942,Y -108.1874,Z 162,A -54.082,B 22.5471,C -0.8776,E1 22.6624,E2 501.4737} C_DIS
LIN {X 87.1592,Y -105.4954,Z 162,A -52.2831,B 22.5469,C -0.8813,E1 22.6663,E2 499.6729} C_DIS
LIN {X 90.3556,Y -102.7715,Z 162,A -50.4979,B 22.5467,C -0.8867,E1 22.67,E2 497.8815} C_DIS
LIN {X 93.4487,Y -99.9669,Z 162,A -48.7806,B 22.5467,C -0.8892,E1 22.6736,E2 496.1656} C_DIS
LIN {X 96.7585,Y -96.7676,Z 162,A -46.8398,B 22.5464,C -0.8945,E1 22.6774,E2 494.22} C_DIS
LIN {X 99.921,Y -93.498,Z 162,A -44.9344,B 22.5463,C -0.8993,E1 22.6811,E2 492.3114} C_DIS
LIN {X 102.8987,Y -90.2105,Z 162,A -43.0955,B 22.5461,C -0.9031,E1 22.6845,E2 490.4719} C_DIS
LIN {X 105.9082,Y -86.657,Z 162,A -41.2263,B 22.5461,C -0.9041,E1 22.6879,E2 488.6099} C_DIS
LIN {X 108.5279,Y -83.3531,Z 162,A -39.418,B 22.5458,C -0.911,E1 22.691,E2 486.7931} C_DIS
LIN {X 111.1107,Y -79.878,Z 162,A -37.6032,B 22.5456,C -0.9161,E1 22.694,E2 484.975} C_DIS
LIN {X 113.301,Y -76.7389,Z 162,A -35.9486,B 22.5453,C -0.9233,E1 22.6966,E2 483.3109} C_DIS
LIN {X 115.2293,Y -73.8118,Z 162,A -34.4405,B 22.5451,C -0.9296,E1 22.6989,E2 481.795} C_DIS
LIN {X 117.9506,Y -69.3804,Z 162,A -32.4302,B 22.5451,C -0.9271,E1 22.7017,E2 479.8026} C_DIS
LIN {X 119.7037,Y -66.31,Z 162,A -30.9241,B 22.545,C -0.9328,E1 22.7038,E2 478.2907} C_DIS
LIN {X 121.7463,Y -62.4778,Z 162,A -29.1844,B 22.545,C -0.9341,E1 22.706,E2 476.5579} C_DIS
LIN {X 123.2098,Y -59.5411,Z 162,A -27.8059,B 22.5447,C -0.9384,E1 22.7077,E2 475.1764} C_DIS
LIN {X 124.8177,Y -56.0895,Z 162,A -25.9113,B 22.5439,C -0.9591,E1 22.71,E2 473.2398} C_DIS
LIN {X 126.3063,Y -52.6515,Z 162,A -24.9026,B 22.5449,C -0.9345,E1 22.711,E2 472.3009} C_DIS
LIN {X 128.0669,Y -48.2119,Z 162,A -22.5834,B 22.544,C -0.9574,E1 22.7134,E2 469.9369} C_DIS
LIN {X 129.7139,Y -43.5881,Z 162,A -20.8819,B 22.5445,C -0.9453,E1 22.7149,E2 468.2775} C_DIS
LIN {X 130.7261,Y -40.4517,Z 162,A -19.2676,B 22.5438,C -0.9619,E1 22.7163,E2 466.6304} C_DIS
LIN {X 131.7813,Y -36.867,Z 162,A -17.7928,B 22.5438,C -0.9622,E1 22.7174,E2 465.1644} C_DIS
LIN {X 132.7364,Y -33.2673,Z 162,A -15.479,B 22.5419,C -1.0069,E1 22.7191,E2 462.7496} C_DIS
LIN {X 134.027,Y -27.6115,Z 162,A -13.8108,B 22.5433,C -0.9745,E1 22.72,E2 461.1762} C_DIS
LIN {X 134.643,Y -24.4315,Z 162,A -12.4601,B 22.5431,C -0.9786,E1 22.7207,E2 459.8238} C_DIS
LIN {X 135.2091,Y -21.0726,Z 162,A -10.7108,B 22.5422,C -1.0002,E1 22.7215,E2 458.03} C_DIS
LIN {X 135.7208,Y -17.4789,Z 162,A -9.3186,B 22.5423,C -0.9984,E1 22.722,E2 456.6517} C_DIS
LIN {X 136.3073,Y -12.0921,Z 162,A -7.1901,B 22.5423,C -0.9984,E1 22.7225,E2 454.5375} C_DIS
LIN {X 136.6033,Y -8.0772,Z 162,A -5.6568,B 22.5424,C -0.9959,E1 22.7228,E2 453.0209} C_DIS
LIN {X 136.8209,Y -2.3776,Z 162,A -2.6324,B 22.5406,C -1.0371,E1 22.723,E2 449.9097} C_DIS
LIN {X 136.8145,Y 2.7625,Z 162,A -1.0217,B 22.5416,C -1.0155,E1 22.723,E2 448.3657} C_DIS
LIN {X 136.517,Y 9.4297,Z 162,A 1.781,B 22.5412,C -1.0249,E1 22.7226,E2 445.5573} C_DIS
LIN {X 136.1407,Y 13.8494,Z 162,A 3.6323,B 22.5409,C -1.0306,E1 22.7221,E2 443.7038} C_DIS
LIN {X 135.5767,Y 18.5774,Z 162,A 5.7623,B 22.5403,C -1.0441,E1 22.7213,E2 441.5529} C_DIS
LIN {X 135.099,Y 21.7798,Z 162,A 6.9338,B 22.5406,C -1.0387,E1 22.7208,E2 440.4029} C_DIS
LIN {X 134.3885,Y 25.7927,Z 162,A 8.5414,B 22.5406,C -1.039,E1 22.72,E2 438.8053} C_DIS
LIN {X 133.5158,Y 29.9881,Z 162,A 10.3208,B 22.5404,C -1.0438,E1 22.7189,E2 437.025} C_DIS
LIN {X 132.6948,Y 33.4311,Z 162,A 11.7808,B 22.5402,C -1.0472,E1 22.718,E2 435.5655} C_DIS
LIN {X 131.8144,Y 36.7486,Z 162,A 13.1879,B 22.5401,C -1.0501,E1 22.7169,E2 434.16} C_DIS
LIN {X 130.6465,Y 40.7075,Z 162,A 15.5635,B 22.5383,C -1.0892,E1 22.7149,E2 431.6982} C_DIS
LIN {X 128.9705,Y 45.7448,Z 162,A 17.1964,B 22.5394,C -1.065,E1 22.7135,E2 430.1384} C_DIS
LIN {X 127.6503,Y 49.3047,Z 162,A 18.787,B 22.5392,C -1.0698,E1 22.7119,E2 428.5454} C_DIS
LIN {X 126.1986,Y 52.9094,Z 162,A 20.3414,B 22.5392,C -1.0708,E1 22.7102,E2 426.9979} C_DIS
LIN {X 124.6267,Y 56.5167,Z 162,A 22.0987,B 22.5387,C -1.0812,E1 22.7082,E2 425.2244} C_DIS
LIN {X 123.0328,Y 59.9072,Z 162,A 23.5017,B 22.5389,C -1.077,E1 22.7065,E2 423.8406} C_DIS
LIN {X 121.4299,Y 63.0917,Z 162,A 25.0634,B 22.5385,C -1.0848,E1 22.7045,E2 422.2681} C_DIS
LIN {X 119.363,Y 66.9214,Z 162,A 26.8919,B 22.5383,C -1.0901,E1 22.7021,E2 420.4365} C_DIS
LIN {X 117.1256,Y 70.7642,Z 162,A 28.7369,B 22.5381,C -1.0943,E1 22.6994,E2 418.5913} C_DIS
LIN {X 114.6889,Y 74.6489,Z 162,A 30.6135,B 22.538,C -1.0971,E1 22.6966,E2 416.7181} C_DIS
LIN {X 112.9125,Y 77.3095,Z 162,A 31.9084,B 22.5379,C -1.0982,E1 22.6946,E2 415.4274} C_DIS
LIN {X 109.8474,Y 81.606,Z 162,A 34.1958,B 22.5375,C -1.1078,E1 22.6908,E2 413.1275} C_DIS
LIN {X 107.0182,Y 85.2824,Z 162,A 36.0824,B 22.5374,C -1.1096,E1 22.6876,E2 411.2461} C_DIS
LIN {X 104.1931,Y 88.7118,Z 162,A 37.9633,B 22.5371,C -1.1151,E1 22.6842,E2 409.3607} C_DIS
LIN {X 100.9159,Y 92.4231,Z 162,A 40.0159,B 22.5369,C -1.1188,E1 22.6804,E2 407.3088} C_DIS
LIN {X 97.9315,Y 95.5798,Z 162,A 41.8521,B 22.5367,C -1.1237,E1 22.6768,E2 405.4688} C_DIS
LIN {X 95.3219,Y 98.1822,Z 162,A 43.3832,B 22.5366,C -1.1264,E1 22.6738,E2 403.9379} C_DIS
LIN {X 92.1131,Y 101.1988,Z 162,A 45.2213,B 22.5364,C -1.1299,E1 22.67,E2 402.099} C_DIS
LIN {X 89.2276,Y 103.7517,Z 162,A 46.7926,B 22.5364,C -1.131,E1 22.6667,E2 400.5319} C_DIS
LIN {X 84.0808,Y 107.9652,Z 162,A 49.5976,B 22.5361,C -1.1372,E1 22.6606,E2 397.7225} C_DIS
LIN {X 80.5848,Y 110.5992,Z 162,A 51.4382,B 22.5359,C -1.1409,E1 22.6565,E2 395.8797} C_DIS
LIN {X 76.8352,Y 113.2358,Z 162,A 53.3375,B 22.5358,C -1.1431,E1 22.6521,E2 393.9819} C_DIS
LIN {X 72.8903,Y 115.8145,Z 162,A 55.2597,B 22.5358,C -1.1437,E1 22.6476,E2 392.0652} C_DIS
LIN {X 69.0742,Y 118.1305,Z 162,A 57.1716,B 22.5355,C -1.1487,E1 22.643,E2 390.147} C_DIS
LIN {X 65.1202,Y 120.3558,Z 162,A 59.0948,B 22.5353,C -1.1525,E1 22.6383,E2 388.2201} C_DIS
LIN {X 61.0852,Y 122.4516,Z 162,A 60.917,B 22.5354,C -1.151,E1 22.6338,E2 386.4075} C_DIS
LIN {X 57.6161,Y 124.1204,Z 162,A 62.4024,B 22.5356,C -1.1467,E1 22.6301,E2 384.9376} C_DIS
LIN {X 53.8409,Y 125.8048,Z 162,A 64.1608,B 22.5355,C -1.15,E1 22.6256,E2 383.1754} C_DIS
LIN {X 49.1076,Y 127.7269,Z 162,A 66.4165,B 22.5351,C -1.158,E1 22.6197,E2 380.9046} C_DIS
LIN {X 45.7278,Y 128.9766,Z 162,A 67.9635,B 22.5349,C -1.1613,E1 22.6156,E2 379.3527} C_DIS
LIN {X 41.8349,Y 130.2895,Z 162,A 69.5989,B 22.535,C -1.1585,E1 22.6113,E2 377.7277} C_DIS
LIN {X 38.2827,Y 131.3771,Z 162,A 71.1009,B 22.5351,C -1.1571,E1 22.6073,E2 376.2325} C_DIS
LIN {X 34.7209,Y 132.3641,Z 162,A 72.7398,B 22.5348,C -1.1626,E1 22.6028,E2 374.5822} C_DIS
LIN {X 30.7995,Y 133.3304,Z 162,A 74.3527,B 22.535,C -1.1598,E1 22.5985,E2 372.9792} C_DIS
LIN {X 27.5446,Y 134.0406,Z 162,A 75.7332,B 22.535,C -1.1598,E1 22.5947,E2 371.6007} C_DIS
LIN {X 18.8072,Y 135.5439,Z 162,A 79.5594,B 22.5346,C -1.1665,E1 22.5841,E2 367.7612} C_DIS
LIN {X 14.6406,Y 136.0559,Z 162,A 80.9803,B 22.5354,C -1.1506,E1 22.5803,E2 366.3831} C_DIS
LIN {X 9.7373,Y 136.4947,Z 162,A 83.866,B 22.5334,C -1.1908,E1 22.572,E2 363.3941} C_DIS
LIN {X 4.6345,Y 136.7647,Z 162,A 85.512,B 22.5346,C -1.1667,E1 22.5676,E2 361.8116} C_DIS
LIN {X 1.3116,Y 136.8364,Z 162,A 87.316,B 22.5337,C -1.1865,E1 22.5624,E2 359.9562} C_DIS
LIN {X -3.2616,Y 136.8037,Z 162,A 89.104,B 22.534,C -1.1798,E1 22.5574,E2 358.1853} C_DIS
LIN {X -7.0809,Y 136.6583,Z 162,A 90.3866,B 22.5348,C -1.164,E1 22.554,E2 356.9437} C_DIS
LIN {X -11.368,Y 136.3685,Z 162,A 91.9554,B 22.5353,C -1.1522,E1 22.5497,E2 355.4048} C_DIS
LIN {X -18.4522,Y 135.5932,Z 162,A 95.1897,B 22.5348,C -1.1625,E1 22.5406,E2 352.1415} C_DIS
LIN {X -22.3691,Y 135.0007,Z 162,A 96.7512,B 22.5351,C -1.1567,E1 22.5364,E2 350.5934} C_DIS
LIN {X -25.7116,Y 134.404,Z 162,A 98.1482,B 22.5352,C -1.1545,E1 22.5325,E2 349.2005} C_DIS
LIN {X -29.0134,Y 133.7302,Z 162,A 99.6517,B 22.5351,C -1.1577,E1 22.5284,E2 347.6867} C_DIS
LIN {X -33.3966,Y 132.7036,Z 162,A 101.4696,B 22.5353,C -1.1528,E1 22.5235,E2 345.8789} C_DIS
LIN {X -36.3516,Y 131.9255,Z 162,A 102.6365,B 22.5356,C -1.1462,E1 22.5204,E2 344.7273} C_DIS
LIN {X -41.7989,Y 130.301,Z 162,A 105.8363,B 22.5339,C -1.1823,E1 22.5116,E2 341.4267} C_DIS
LIN {X -46.9746,Y 128.5271,Z 162,A 107.191,B 22.5362,C -1.1353,E1 22.5084,E2 340.1921} C_DIS
LIN {X -52.8551,Y 126.2212,Z 162,A 109.8766,B 22.5362,C -1.1335,E1 22.5014,E2 337.5045} C_DIS
LIN {X -55.5725,Y 125.049,Z 162,A 111.3569,B 22.5358,C -1.143,E1 22.4975,E2 335.9956} C_DIS
LIN {X -58.7649,Y 123.5807,Z 162,A 112.749,B 22.5361,C -1.137,E1 22.494,E2 334.6151} C_DIS
LIN {X -61.6085,Y 122.1888,Z 162,A 114.1964,B 22.5359,C -1.1406,E1 22.4904,E2 333.154} C_DIS
LIN {X -69.0041,Y 118.1717,Z 162,A 117.8116,B 22.5359,C -1.1387,E1 22.4815,E2 329.5322} C_DIS
LIN {X -72.0635,Y 116.331,Z 162,A 119.5056,B 22.5357,C -1.1452,E1 22.4774,E2 327.8151} C_DIS
LIN {X -74.953,Y 114.4908,Z 162,A 120.5691,B 22.5366,C -1.1253,E1 22.4751,E2 326.8} C_DIS
LIN {X -77.0025,Y 113.1226,Z 162,A 121.8055,B 22.5363,C -1.1327,E1 22.4721,E2 325.5395} C_DIS
LIN {X -80.766,Y 110.4668,Z 162,A 123.7256,B 22.5365,C -1.1284,E1 22.4678,E2 323.6232} C_DIS
LIN {X -83.4567,Y 108.4487,Z 162,A 125.1312,B 22.5366,C -1.1253,E1 22.4647,E2 322.22} C_DIS
LIN {X -86.8563,Y 105.7453,Z 162,A 126.963,B 22.5368,C -1.122,E1 22.4607,E2 320.3892} C_DIS
LIN {X -90.1212,Y 102.9766,Z 162,A 128.7539,B 22.537,C -1.1179,E1 22.4569,E2 318.6012} C_DIS
LIN {X -93.536,Y 99.8856,Z 162,A 130.694,B 22.5372,C -1.1139,E1 22.4529,E2 316.6626} C_DIS
LIN {X -96.7902,Y 96.7357,Z 162,A 132.6196,B 22.5373,C -1.1107,E1 22.4491,E2 314.7362} C_DIS
LIN {X -99.9356,Y 93.4824,Z 162,A 134.5108,B 22.5375,C -1.1059,E1 22.4455,E2 312.8485} C_DIS
LIN {X -102.9362,Y 90.1675,Z 162,A 136.2455,B 22.5381,C -1.0949,E1 22.4423,E2 311.1339} C_DIS
LIN {X -104.6486,Y 88.1744,Z 162,A 137.3779,B 22.5381,C -1.0935,E1 22.4402,E2 309.9994} C_DIS
LIN {X -107.4332,Y 84.7595,Z 162,A 139.0375,B 22.5387,C -1.0802,E1 22.4374,E2 308.3659} C_DIS
LIN {X -109.9066,Y 81.5265,Z 162,A 141.0503,B 22.5383,C -1.0897,E1 22.4339,E2 306.3175} C_DIS
LIN {X -113.4619,Y 76.5005,Z 162,A 143.5659,B 22.5387,C -1.0797,E1 22.4299,E2 303.814} C_DIS
LIN {X -115.7552,Y 72.9844,Z 162,A 145.4079,B 22.5387,C -1.0786,E1 22.4271,E2 301.9646} C_DIS
LIN {X -118.1224,Y 69.0879,Z 162,A 147.178,B 22.5393,C -1.0668,E1 22.4246,E2 300.215} C_DIS
LIN {X -121.2065,Y 63.5171,Z 162,A 149.9078,B 22.5395,C -1.0619,E1 22.421,E2 297.482} C_DIS
LIN {X -122.6715,Y 60.6394,Z 162,A 151.1531,B 22.5399,C -1.0531,E1 22.4194,E2 296.2524} C_DIS
LIN {X -123.9934,Y 57.8906,Z 162,A 152.6285,B 22.5397,C -1.0582,E1 22.4176,E2 294.7546} C_DIS
LIN {X -125.4388,Y 54.6874,Z 162,A 153.8951,B 22.5403,C -1.0445,E1 22.4162,E2 293.5161} C_DIS
LIN {X -127.367,Y 50.0334,Z 162,A 156.1464,B 22.5403,C -1.0445,E1 22.4139,E2 291.2509} C_DIS
LIN {X -128.5386,Y 46.9425,Z 162,A 157.6844,B 22.5403,C -1.0471,E1 22.4123,E2 289.6962} C_DIS
LIN {X -129.7817,Y 43.3843,Z 162,A 159.2441,B 22.5405,C -1.0413,E1 22.4109,E2 288.1415} C_DIS
LIN {X -131.0235,Y 39.4799,Z 162,A 161.0333,B 22.5405,C -1.0393,E1 22.4095,E2 286.3463} C_DIS
Enddeposition()
END
